C07310=1132.856,310.921,-76.435,-177.796,10.546,149.531
C07311=1132.851,311.169,-76.468,-177.793,10.548,149.531
C07312=1132.848,311.417,-76.500,-177.790,10.550,149.530
C07313=1132.844,311.665,-76.533,-177.787,10.553,149.530
C07314=1132.839,311.913,-76.564,-177.783,10.556,149.530
C07315=1132.835,312.160,-76.597,-177.780,10.558,149.530
C07316=1132.831,312.408,-76.629,-177.777,10.561,149.530
C07317=1132.827,312.656,-76.662,-177.774,10.563,149.529
C07318=1132.824,312.904,-76.694,-177.771,10.566,149.529
C07319=1132.820,313.152,-76.727,-177.767,10.569,149.529
C07320=1132.815,313.400,-76.760,-177.765,10.571,149.529
C07321=1132.812,313.648,-76.792,-177.761,10.574,149.529
C07322=1132.807,313.895,-76.824,-177.758,10.576,149.529
C07323=1132.803,314.143,-76.857,-177.755,10.579,149.529
C07324=1132.799,314.391,-76.889,-177.752,10.581,149.528
C07325=1132.795,314.639,-76.923,-177.749,10.584,149.528
C07326=1132.791,314.887,-76.954,-177.745,10.587,149.528
C07327=1132.787,315.134,-76.988,-177.742,10.589,149.528
C07328=1132.782,315.383,-77.020,-177.739,10.592,149.528
C07329=1132.779,315.630,-77.053,-177.736,10.594,149.527
C07330=1132.775,315.878,-77.086,-177.733,10.596,149.527
C07331=1132.770,316.126,-77.118,-177.730,10.599,149.527
C07332=1132.767,316.374,-77.151,-177.727,10.601,149.527
C07333=1132.763,316.621,-77.184,-177.724,10.604,149.527
C07334=1132.758,316.870,-77.216,-177.721,10.606,149.526
C07335=1132.754,317.118,-77.249,-177.717,10.609,149.526
C07336=1132.751,317.365,-77.282,-177.714,10.612,149.526
C07337=1132.746,317.613,-77.314,-177.711,10.614,149.526
C07338=1132.742,317.861,-77.348,-177.708,10.616,149.526
C07339=1132.738,318.109,-77.381,-177.705,10.619,149.525
C07340=1132.735,318.356,-77.413,-177.701,10.622,149.525
C07341=1132.730,318.605,-77.446,-177.698,10.624,149.525
C07342=1132.726,318.852,-77.479,-177.695,10.627,149.525
C07343=1132.722,319.100,-77.512,-177.692,10.629,149.525
C07344=1132.719,319.347,-77.545,-177.689,10.632,149.525
C07345=1132.714,319.595,-77.578,-177.686,10.635,149.524
C07346=1132.710,319.843,-77.611,-177.682,10.637,149.524
C07347=1132.706,320.091,-77.643,-177.679,10.640,149.524
C07348=1132.702,320.339,-77.677,-177.676,10.642,149.524
C07349=1132.698,320.587,-77.710,-177.673,10.645,149.524
C07350=1132.695,320.799,-77.738,-177.670,10.647,149.523
C07351=1132.691,321.013,-77.766,-177.668,10.648,149.523
C07352=1132.687,321.226,-77.794,-177.665,10.651,149.523
C07353=1132.684,321.440,-77.824,-177.662,10.653,149.523
C07354=1132.680,321.653,-77.852,-177.659,10.655,149.523
C07355=1132.677,321.866,-77.881,-177.657,10.657,149.523
C07356=1132.673,322.080,-77.909,-177.654,10.659,149.522
C07357=1132.671,322.293,-77.937,-177.651,10.662,149.522
C07358=1132.667,322.541,-77.971,-177.648,10.664,149.522
C07359=1132.663,322.788,-78.004,-177.645,10.667,149.522
C07360=1132.658,323.036,-78.037,-177.642,10.670,149.522
C07361=1132.654,323.284,-78.070,-177.638,10.672,149.521
C07362=1132.650,323.532,-78.103,-177.635,10.675,149.521
C07363=1132.646,323.779,-78.136,-177.632,10.677,149.521
C07364=1132.642,324.027,-78.170,-177.629,10.680,149.521
C07365=1132.638,324.276,-78.203,-177.625,10.682,149.521
C07366=1132.634,324.523,-78.236,-177.623,10.684,149.521
C07367=1132.630,324.770,-78.270,-177.620,10.687,149.520
C07368=1132.626,325.018,-78.303,-177.616,10.689,149.520
C07369=1132.622,325.266,-78.336,-177.614,10.692,149.520
C07370=1132.618,325.514,-78.370,-177.610,10.694,149.520
C07371=1132.614,325.761,-78.403,-177.607,10.697,149.520
C07372=1132.610,326.010,-78.436,-177.604,10.699,149.519
C07373=1132.606,326.257,-78.470,-177.601,10.702,149.519
C07374=1132.602,326.505,-78.503,-177.597,10.704,149.519
C07375=1132.598,326.752,-78.536,-177.594,10.707,149.519
C07376=1132.594,327.000,-78.570,-177.591,10.710,149.519
C07377=1132.590,327.247,-78.603,-177.588,10.712,149.518
C07378=1132.586,327.496,-78.638,-177.584,10.714,149.518
C07379=1132.582,327.744,-78.671,-177.582,10.717,149.518
C07380=1132.578,327.991,-78.705,-177.578,10.720,149.518
C07381=1132.574,328.238,-78.738,-177.575,10.722,149.518
C07382=1132.570,328.486,-78.771,-177.572,10.725,149.518
C07383=1132.566,328.734,-78.805,-177.569,10.727,149.517
C07384=1132.562,328.982,-78.838,-177.565,10.730,149.517
C07385=1132.557,329.230,-78.872,-177.562,10.732,149.517
C07386=1132.554,329.477,-78.906,-177.559,10.735,149.517
C07387=1132.550,329.725,-78.939,-177.556,10.737,149.516
C07388=1132.546,329.972,-78.973,-177.552,10.740,149.516
C07389=1132.542,330.220,-79.007,-177.549,10.743,149.516
C07390=1132.538,330.467,-79.040,-177.546,10.745,149.516
C07391=1132.534,330.716,-79.074,-177.543,10.748,149.516
C07392=1132.530,330.963,-79.108,-177.540,10.749,149.515
C07393=1132.526,331.211,-79.142,-177.537,10.752,149.515
C07394=1132.522,331.458,-79.175,-177.534,10.754,149.515
C07395=1132.518,331.707,-79.210,-177.531,10.757,149.515
C07396=1132.514,331.954,-79.243,-177.527,10.759,149.515
C07397=1132.510,332.202,-79.277,-177.524,10.762,149.515
C07398=1132.507,332.449,-79.311,-177.521,10.765,149.514
C07399=1132.502,332.697,-79.345,-177.518,10.767,149.514
C07400=1132.498,332.944,-79.378,-177.514,10.769,149.514
C07401=1132.495,333.192,-79.413,-177.511,10.772,149.514
C07402=1132.490,333.440,-79.446,-177.508,10.775,149.514
C07403=1132.486,333.687,-79.480,-177.505,10.777,149.513
C07404=1132.483,333.935,-79.514,-177.501,10.780,149.513
C07405=1132.478,334.183,-79.548,-177.499,10.782,149.513
C07406=1132.474,334.396,-79.577,-177.496,10.784,149.513
C07407=1132.472,334.609,-79.607,-177.493,10.787,149.513
C07408=1132.468,334.822,-79.636,-177.490,10.789,149.512
C07409=1132.465,335.036,-79.666,-177.487,10.791,149.512
C07410=1132.461,335.249,-79.695,-177.485,10.793,149.512
C07411=1132.458,335.462,-79.724,-177.481,10.795,149.512
C07412=1132.454,335.676,-79.753,-177.479,10.797,149.512
C07413=1132.450,335.888,-79.782,-177.476,10.799,149.511
C07414=1132.447,336.136,-79.817,-177.473,10.802,149.511
C07415=1132.443,336.384,-79.851,-177.470,10.804,149.511
C07416=1132.439,336.632,-79.885,-177.467,10.807,149.511
C07417=1132.435,336.879,-79.920,-177.463,10.809,149.511
C07418=1132.431,337.126,-79.954,-177.460,10.812,149.510
C07419=1132.427,337.374,-79.987,-177.457,10.814,149.510
C07420=1132.423,337.622,-80.022,-177.454,10.817,149.510
C07421=1132.420,337.870,-80.056,-177.451,10.819,149.510
C07422=1132.415,338.117,-80.090,-177.447,10.822,149.510
C07423=1132.412,338.365,-80.125,-177.444,10.825,149.510
C07424=1132.407,338.612,-80.159,-177.441,10.827,149.509
C07425=1132.403,338.859,-80.193,-177.438,10.830,149.509
C07426=1132.400,339.108,-80.228,-177.434,10.832,149.509
C07427=1132.396,339.355,-80.262,-177.431,10.834,149.509
C07428=1132.392,339.603,-80.296,-177.428,10.837,149.508
C07429=1132.387,339.850,-80.331,-177.425,10.840,149.508
C07430=1132.384,340.098,-80.365,-177.422,10.842,149.508
C07431=1132.379,340.345,-80.400,-177.418,10.845,149.508
C07432=1132.376,340.593,-80.434,-177.415,10.847,149.508
C07433=1132.372,340.841,-80.468,-177.412,10.849,149.507
C07434=1132.368,341.088,-80.502,-177.409,10.852,149.507
C07435=1132.364,341.336,-80.537,-177.405,10.855,149.507
C07436=1132.359,341.583,-80.571,-177.402,10.857,149.507
C07437=1132.356,341.831,-80.606,-177.399,10.860,149.507
C07438=1132.352,342.078,-80.641,-177.395,10.862,149.506
C07439=1132.348,342.326,-80.676,-177.392,10.865,149.506
C07440=1132.344,342.573,-80.710,-177.389,10.867,149.506
C07441=1132.340,342.821,-80.744,-177.386,10.870,149.506
C07442=1132.335,343.069,-80.779,-177.383,10.872,149.506
C07443=1132.332,343.316,-80.814,-177.379,10.875,149.506
C07444=1132.328,343.564,-80.849,-177.377,10.876,149.505
C07445=1132.324,343.811,-80.883,-177.373,10.879,149.505
C07446=1132.321,344.059,-80.917,-177.370,10.882,149.505
C07447=1132.316,344.306,-80.953,-177.367,10.884,149.505
C07448=1132.312,344.554,-80.987,-177.364,10.887,149.505
C07449=1132.308,344.802,-81.022,-177.360,10.889,149.504
C07450=1132.305,345.049,-81.057,-177.357,10.891,149.504
C07451=1132.300,345.296,-81.091,-177.354,10.894,149.504
C07452=1132.296,345.544,-81.126,-177.350,10.896,149.504
C07453=1132.293,345.792,-81.162,-177.348,10.899,149.504
C07454=1132.289,346.039,-81.196,-177.344,10.902,149.503
C07455=1132.285,346.287,-81.230,-177.341,10.904,149.503
C07456=1132.281,346.534,-81.266,-177.338,10.907,149.503
C07457=1132.277,346.782,-81.300,-177.334,10.909,149.503
C07458=1132.273,347.030,-81.336,-177.331,10.911,149.502
C07459=1132.269,347.277,-81.370,-177.328,10.914,149.502
C07460=1132.266,347.524,-81.405,-177.324,10.916,149.502
C07461=1132.262,347.772,-81.440,-177.321,10.919,149.502
C07462=1132.258,347.985,-81.470,-177.319,10.921,149.502
C07463=1132.255,348.198,-81.500,-177.315,10.923,149.501
C07464=1132.251,348.412,-81.530,-177.313,10.925,149.501
C07465=1132.247,348.624,-81.560,-177.310,10.928,149.501
C07466=1132.244,348.838,-81.591,-177.307,10.929,149.501
C07467=1132.241,349.050,-81.621,-177.304,10.932,149.501
C07468=1132.237,349.263,-81.651,-177.302,10.934,149.501
C07469=1132.234,349.476,-81.682,-177.299,10.936,149.500
C07470=1132.230,349.724,-81.716,-177.295,10.939,149.500
C07471=1132.227,349.971,-81.751,-177.292,10.941,149.500
C07472=1132.223,350.218,-81.787,-177.288,10.945,149.500
C07473=1132.219,350.467,-81.821,-177.284,10.947,149.499
C07474=1132.215,350.713,-81.857,-177.280,10.950,149.499
C07475=1132.211,350.961,-81.892,-177.277,10.952,149.499
C07476=1132.207,351.209,-81.927,-177.273,10.956,149.499
C07477=1132.203,351.456,-81.963,-177.269,10.958,149.498
C07478=1132.199,351.703,-81.998,-177.266,10.960,149.498
C07479=1132.195,351.951,-82.033,-177.262,10.963,149.498
C07480=1132.192,352.199,-82.068,-177.258,10.966,149.497
C07481=1132.187,352.446,-82.103,-177.255,10.968,149.497
C07482=1132.184,352.693,-82.139,-177.251,10.971,149.497
C07483=1132.180,352.941,-82.174,-177.248,10.974,149.497
C07484=1132.176,353.189,-82.209,-177.243,10.977,149.496
C07485=1132.172,353.436,-82.245,-177.240,10.979,149.496
C07486=1132.168,353.683,-82.280,-177.237,10.982,149.496
C07487=1132.164,353.931,-82.315,-177.233,10.984,149.495
C07488=1132.161,354.178,-82.351,-177.229,10.987,149.495
C07489=1132.157,354.426,-82.387,-177.226,10.989,149.495
C07490=1132.152,354.673,-82.422,-177.222,10.992,149.495
C07491=1132.148,354.920,-82.458,-177.218,10.995,149.494
C07492=1132.145,355.168,-82.493,-177.215,10.997,149.494
C07493=1132.141,355.415,-82.529,-177.211,11.000,149.494
C07494=1132.137,355.663,-82.565,-177.208,11.002,149.494
C07495=1132.134,355.910,-82.600,-177.204,11.004,149.493
C07496=1132.129,356.157,-82.635,-177.200,11.008,149.493
C07497=1132.126,356.405,-82.671,-177.197,11.010,149.493
C07498=1132.121,356.652,-82.707,-177.193,11.012,149.493
C07499=1132.118,356.900,-82.743,-177.190,11.015,149.492
C07500=1132.114,357.147,-82.778,-177.187,11.017,149.492
C07501=1132.110,357.395,-82.814,-177.182,11.020,149.492
C07502=1132.107,357.642,-82.849,-177.179,11.022,149.492
C07503=1132.102,357.890,-82.885,-177.176,11.025,149.491
C07504=1132.098,358.137,-82.920,-177.172,11.027,149.491
C07505=1132.094,358.384,-82.956,-177.169,11.030,149.491
C07506=1132.091,358.631,-82.992,-177.166,11.032,149.491
C07507=1132.087,358.879,-83.028,-177.162,11.034,149.490
C07508=1132.083,359.127,-83.064,-177.158,11.037,149.490
C07509=1132.079,359.374,-83.100,-177.155,11.039,149.490
C07510=1132.076,359.622,-83.135,-177.151,11.042,149.489
C07511=1132.072,359.869,-83.172,-177.148,11.044,149.489
C07512=1132.068,360.116,-83.207,-177.144,11.047,149.489
C07513=1132.064,360.364,-83.243,-177.141,11.049,149.489
C07514=1132.061,360.611,-83.279,-177.138,11.052,149.488
C07515=1132.057,360.859,-83.315,-177.134,11.054,149.488
C07516=1132.053,361.106,-83.351,-177.131,11.056,149.488
C07517=1132.049,361.353,-83.387,-177.127,11.059,149.488
C07518=1132.045,361.566,-83.418,-177.125,11.061,149.487
C07519=1132.042,361.778,-83.449,-177.121,11.063,149.487
C07520=1132.038,361.992,-83.480,-177.119,11.065,149.487
C07521=1132.035,362.204,-83.511,-177.115,11.067,149.487
C07522=1132.032,362.418,-83.542,-177.113,11.069,149.486
C07523=1132.029,362.630,-83.573,-177.110,11.071,149.486
C07524=1132.026,362.843,-83.604,-177.107,11.073,149.486
C07525=1132.023,363.056,-83.635,-177.104,11.075,149.486
C07526=1132.018,363.303,-83.672,-177.101,11.078,149.486
C07527=1132.015,363.551,-83.707,-177.097,11.080,149.485
C07528=1132.011,363.798,-83.744,-177.094,11.082,149.485
C07529=1132.007,364.046,-83.780,-177.091,11.085,149.485
C07530=1132.004,364.293,-83.816,-177.088,11.087,149.485
C07531=1131.999,364.540,-83.852,-177.084,11.090,149.484
C07532=1131.996,364.787,-83.888,-177.081,11.092,149.484
C07533=1131.992,365.035,-83.924,-177.078,11.093,149.484
C07534=1131.988,365.282,-83.961,-177.075,11.096,149.484
C07535=1131.984,365.529,-83.998,-177.071,11.098,149.483
C07536=1131.980,365.777,-84.033,-177.068,11.101,149.483
C07537=1131.976,366.024,-84.070,-177.065,11.103,149.483
C07538=1131.973,366.272,-84.106,-177.061,11.106,149.483
C07539=1131.969,366.519,-84.143,-177.058,11.108,149.482
C07540=1131.966,366.766,-84.179,-177.055,11.110,149.482
C07541=1131.961,367.014,-84.215,-177.052,11.112,149.482
C07542=1131.958,367.261,-84.251,-177.049,11.115,149.482
C07543=1131.954,367.508,-84.288,-177.045,11.117,149.482
C07544=1131.951,367.755,-84.325,-177.042,11.120,149.481
C07545=1131.946,368.003,-84.361,-177.039,11.121,149.481
C07546=1131.942,368.250,-84.398,-177.036,11.124,149.481
C07547=1131.939,368.497,-84.434,-177.032,11.126,149.481
C07548=1131.935,368.744,-84.471,-177.029,11.129,149.480
C07549=1131.932,368.992,-84.507,-177.026,11.131,149.480
C07550=1131.927,369.239,-84.543,-177.023,11.133,149.480
C07551=1131.923,369.486,-84.580,-177.020,11.136,149.480
C07552=1131.920,369.733,-84.617,-177.017,11.138,149.480
C07553=1131.916,369.981,-84.653,-177.014,11.141,149.479
C07554=1131.912,370.228,-84.690,-177.011,11.142,149.479
C07555=1131.908,370.475,-84.726,-177.008,11.145,149.479
C07556=1131.905,370.723,-84.763,-177.004,11.147,149.479
C07557=1131.901,370.970,-84.800,-177.002,11.149,149.478
C07558=1131.897,371.217,-84.836,-176.998,11.151,149.478
C07559=1131.893,371.464,-84.873,-176.995,11.154,149.478
C07560=1131.889,371.712,-84.910,-176.992,11.156,149.478
C07561=1131.886,371.958,-84.946,-176.989,11.158,149.478
C07562=1131.882,372.206,-84.983,-176.986,11.161,149.478
C07563=1131.878,372.454,-85.020,-176.984,11.163,149.477
C07564=1131.874,372.701,-85.057,-176.980,11.165,149.477
C07565=1131.871,372.948,-85.093,-176.977,11.167,149.477
C07566=1131.867,373.195,-85.130,-176.974,11.169,149.477
C07567=1131.863,373.443,-85.167,-176.971,11.172,149.477
C07568=1131.859,373.690,-85.204,-176.968,11.174,149.476
C07569=1131.856,373.937,-85.241,-176.965,11.176,149.476
C07570=1131.852,374.184,-85.277,-176.962,11.179,149.476
C07571=1131.848,374.432,-85.315,-176.959,11.181,149.476
C07572=1131.844,374.679,-85.352,-176.957,11.183,149.476
C07573=1131.840,374.926,-85.388,-176.953,11.186,149.476
C07574=1131.837,375.138,-85.420,-176.951,11.188,149.475
C07575=1131.833,375.351,-85.452,-176.948,11.189,149.475
C07576=1131.830,375.564,-85.484,-176.946,11.191,149.475
C07577=1131.827,375.778,-85.516,-176.944,11.193,149.475
C07578=1131.824,375.990,-85.548,-176.941,11.195,149.475
C07579=1131.821,376.203,-85.580,-176.939,11.197,149.475
C07580=1131.818,376.415,-85.611,-176.937,11.199,149.475
C07581=1131.814,376.628,-85.643,-176.934,11.201,149.475
C07582=1131.811,376.874,-85.680,-176.931,11.204,149.474
C07583=1131.807,377.122,-85.717,-176.928,11.206,149.474
C07584=1131.803,377.370,-85.754,-176.925,11.208,149.474
C07585=1131.799,377.616,-85.791,-176.922,11.211,149.474
C07586=1131.796,377.864,-85.829,-176.920,11.213,149.474
C07587=1131.792,378.111,-85.865,-176.917,11.215,149.474
C07588=1131.788,378.358,-85.902,-176.914,11.217,149.474
C07589=1131.784,378.605,-85.940,-176.911,11.220,149.474
C07590=1131.780,378.853,-85.977,-176.909,11.222,149.473
C07591=1131.776,379.100,-86.014,-176.905,11.224,149.473
C07592=1131.772,379.347,-86.052,-176.903,11.226,149.473
C07593=1131.769,379.594,-86.089,-176.900,11.229,149.473
C07594=1131.765,379.842,-86.126,-176.898,11.231,149.473
C07595=1131.761,380.088,-86.163,-176.895,11.234,149.473
C07596=1131.758,380.336,-86.200,-176.892,11.236,149.473
C07597=1131.755,380.582,-86.237,-176.889,11.238,149.473
C07598=1131.750,380.830,-86.274,-176.887,11.240,149.473
C07599=1131.747,381.077,-86.311,-176.884,11.243,149.473
C07600=1131.742,381.324,-86.350,-176.882,11.245,149.473
C07601=1131.739,381.572,-86.387,-176.878,11.247,149.472
C07602=1131.735,381.819,-86.424,-176.876,11.249,149.472
C07603=1131.731,382.066,-86.461,-176.873,11.252,149.472
C07604=1131.728,382.313,-86.499,-176.871,11.254,149.472
C07605=1131.724,382.560,-86.536,-176.868,11.257,149.472
C07606=1131.720,382.807,-86.574,-176.866,11.259,149.472
C07607=1131.716,383.055,-86.611,-176.863,11.261,149.472
C07608=1131.713,383.301,-86.648,-176.861,11.264,149.472
C07609=1131.710,383.549,-86.686,-176.858,11.266,149.472
C07610=1131.705,383.796,-86.723,-176.857,11.268,149.472
C07611=1131.702,384.043,-86.761,-176.856,11.269,149.472
C07612=1131.698,384.290,-86.798,-176.855,11.271,149.472
C07613=1131.694,384.537,-86.836,-176.853,11.272,149.472
C07614=1131.691,384.785,-86.873,-176.852,11.274,149.473
C07615=1131.687,385.031,-86.910,-176.851,11.276,149.473
C07616=1131.683,385.279,-86.949,-176.850,11.277,149.473
C07617=1131.679,385.526,-86.986,-176.849,11.279,149.473
C07618=1131.675,385.773,-87.023,-176.848,11.281,149.473
C07619=1131.672,386.021,-87.061,-176.847,11.282,149.473
C07620=1131.668,386.267,-87.098,-176.846,11.284,149.474
C07621=1131.665,386.515,-87.136,-176.845,11.286,149.474
C07622=1131.661,386.762,-87.173,-176.844,11.288,149.474
C07623=1131.658,387.009,-87.211,-176.842,11.289,149.474
C07624=1131.654,387.256,-87.249,-176.842,11.291,149.474
C07625=1131.649,387.504,-87.286,-176.841,11.293,149.475
C07626=1131.646,387.750,-87.324,-176.839,11.295,149.475
C07627=1131.642,387.997,-87.362,-176.839,11.297,149.475
C07628=1131.638,388.245,-87.399,-176.838,11.298,149.475
C07629=1131.635,388.491,-87.436,-176.837,11.300,149.475
C07630=1131.632,388.704,-87.469,-176.836,11.302,149.476
C07631=1131.628,388.917,-87.502,-176.835,11.304,149.476
C07632=1131.625,389.129,-87.533,-176.834,11.306,149.476
C07633=1131.622,389.342,-87.566,-176.834,11.307,149.476
C07634=1131.619,389.555,-87.599,-176.833,11.309,149.477
C07635=1131.615,389.767,-87.631,-176.832,11.311,149.477
C07636=1131.613,389.979,-87.663,-176.831,11.313,149.477
C07637=1131.609,390.193,-87.695,-176.831,11.314,149.477
C07638=1131.606,390.439,-87.733,-176.829,11.316,149.478
C07639=1131.602,390.687,-87.772,-176.829,11.318,149.478
C07640=1131.598,390.934,-87.809,-176.828,11.320,149.478
C07641=1131.594,391.181,-87.846,-176.827,11.322,149.479
C07642=1131.591,391.428,-87.884,-176.827,11.325,149.479
C07643=1131.588,391.675,-87.922,-176.826,11.327,149.479
C07644=1131.584,391.922,-87.959,-176.825,11.329,149.480
C07645=1131.579,392.170,-87.997,-176.825,11.331,149.480
C07646=1131.576,392.417,-88.035,-176.824,11.333,149.481
C07647=1131.573,392.664,-88.073,-176.824,11.335,149.481
C07648=1131.569,392.910,-88.110,-176.823,11.337,149.481
C07649=1131.566,393.158,-88.148,-176.822,11.340,149.482
C07650=1131.561,393.405,-88.186,-176.821,11.342,149.482
C07651=1131.557,393.652,-88.223,-176.821,11.344,149.483
C07652=1131.554,393.899,-88.261,-176.820,11.347,149.483
C07653=1131.550,394.146,-88.299,-176.820,11.349,149.484
C07654=1131.546,394.393,-88.337,-176.819,11.351,149.484
C07655=1131.542,394.640,-88.375,-176.819,11.353,149.485
C07656=1131.539,394.888,-88.412,-176.818,11.356,149.485
C07657=1131.536,395.135,-88.450,-176.817,11.359,149.486
C07658=1131.531,395.382,-88.488,-176.817,11.361,149.486
C07659=1131.528,395.629,-88.526,-176.817,11.363,149.487
C07660=1131.524,395.876,-88.564,-176.816,11.366,149.487
C07661=1131.520,396.123,-88.602,-176.816,11.368,149.488
C07662=1131.516,396.370,-88.640,-176.816,11.370,149.488
C07663=1131.513,396.617,-88.678,-176.815,11.374,149.489
C07664=1131.509,396.864,-88.715,-176.815,11.376,149.489
C07665=1131.505,397.112,-88.753,-176.815,11.379,149.490
C07666=1131.501,397.358,-88.791,-176.815,11.381,149.491
C07667=1131.498,397.606,-88.829,-176.814,11.383,149.491
C07668=1131.494,397.852,-88.866,-176.814,11.386,149.492
C07669=1131.490,398.100,-88.905,-176.813,11.389,149.493
C07670=1131.487,398.346,-88.942,-176.813,11.392,149.493
C07671=1131.483,398.594,-88.980,-176.813,11.394,149.494
C07672=1131.479,398.841,-89.019,-176.813,11.397,149.495
C07673=1131.476,399.088,-89.056,-176.813,11.399,149.495
C07674=1131.472,399.334,-89.094,-176.812,11.403,149.496
C07675=1131.468,399.582,-89.133,-176.813,11.406,149.497
C07676=1131.465,399.829,-89.171,-176.813,11.408,149.497
C07677=1131.461,400.076,-89.208,-176.813,11.411,149.498
C07678=1131.457,400.323,-89.247,-176.812,11.414,149.499
C07679=1131.453,400.570,-89.284,-176.812,11.417,149.499
C07680=1131.450,400.817,-89.322,-176.812,11.420,149.500
C07681=1131.445,401.065,-89.360,-176.812,11.422,149.501
C07682=1131.442,401.312,-89.398,-176.812,11.426,149.502
C07683=1131.438,401.559,-89.435,-176.812,11.429,149.502
C07684=1131.434,401.806,-89.474,-176.812,11.432,149.503
C07685=1131.432,402.053,-89.512,-176.812,11.435,149.504
C07686=1131.428,402.265,-89.545,-176.812,11.438,149.505
C07687=1131.425,402.478,-89.577,-176.812,11.441,149.506
C07688=1131.422,402.691,-89.610,-176.812,11.443,149.506
C07689=1131.419,402.903,-89.642,-176.813,11.446,149.507
C07690=1131.415,403.115,-89.675,-176.812,11.449,149.508
C07691=1131.413,403.328,-89.708,-176.813,11.452,149.509
C07692=1131.409,403.540,-89.741,-176.813,11.454,149.509
C07693=1131.406,403.753,-89.773,-176.813,11.457,149.510
C07694=1131.402,404.000,-89.811,-176.813,11.460,149.511
C07695=1131.399,404.248,-89.850,-176.814,11.463,149.512
C07696=1131.395,404.494,-89.887,-176.814,11.467,149.513
C07697=1131.391,404.742,-89.926,-176.814,11.470,149.514
C07698=1131.387,404.988,-89.963,-176.815,11.473,149.515
C07699=1131.384,405.236,-90.001,-176.815,11.477,149.516
C07700=1131.380,405.482,-90.040,-176.816,11.480,149.517
C07701=1131.376,405.729,-90.078,-176.816,11.483,149.518
C07702=1131.373,405.976,-90.116,-176.816,11.487,149.519
C07703=1131.369,406.223,-90.154,-176.817,11.490,149.520
C07704=1131.366,406.471,-90.192,-176.817,11.494,149.521
C07705=1131.361,406.717,-90.230,-176.817,11.497,149.522
C07706=1131.358,406.965,-90.268,-176.818,11.502,149.523
C07707=1131.355,407.212,-90.306,-176.819,11.505,149.524
C07708=1131.350,407.459,-90.344,-176.819,11.508,149.525
C07709=1131.347,407.706,-90.382,-176.819,11.512,149.526
C07710=1131.343,407.953,-90.422,-176.820,11.516,149.527
C07711=1131.340,408.200,-90.459,-176.821,11.520,149.528
C07712=1131.336,408.447,-90.497,-176.822,11.523,149.529
C07713=1131.332,408.694,-90.535,-176.822,11.527,149.531
C07714=1131.329,408.941,-90.573,-176.823,11.531,149.532
C07715=1131.325,409.189,-90.612,-176.823,11.535,149.533
C07716=1131.321,409.435,-90.649,-176.824,11.539,149.534
C07717=1131.317,409.682,-90.689,-176.824,11.543,149.535
C07718=1131.314,409.929,-90.726,-176.825,11.546,149.536
C07719=1131.310,410.176,-90.764,-176.826,11.551,149.538
C07720=1131.306,410.424,-90.803,-176.826,11.555,149.539
C07721=1131.303,410.670,-90.840,-176.828,11.559,149.540
C07722=1131.299,410.917,-90.879,-176.828,11.563,149.542
C07723=1131.296,411.164,-90.917,-176.829,11.567,149.543
C07724=1131.291,411.411,-90.955,-176.830,11.571,149.544
C07725=1131.288,411.659,-90.993,-176.831,11.575,149.545
C07726=1131.284,411.906,-91.032,-176.832,11.579,149.547
C07727=1131.281,412.152,-91.070,-176.833,11.584,149.548
C07728=1131.277,412.400,-91.109,-176.834,11.588,149.549
C07729=1131.274,412.647,-91.147,-176.835,11.592,149.551
C07730=1131.270,412.893,-91.184,-176.836,11.596,149.552
C07731=1131.266,413.141,-91.223,-176.837,11.600,149.553
C07732=1131.262,413.387,-91.261,-176.838,11.605,149.555
C07733=1131.258,413.635,-91.300,-176.839,11.609,149.556
C07734=1131.255,413.882,-91.338,-176.840,11.614,149.558
C07735=1131.251,414.129,-91.376,-176.841,11.619,149.559
C07736=1131.248,414.375,-91.414,-176.842,11.623,149.561
C07737=1131.246,414.623,-91.452,-176.844,11.627,149.562
C07738=1131.243,414.870,-91.491,-176.845,11.632,149.564
C07739=1131.242,415.117,-91.528,-176.846,11.637,149.565
C07740=1131.242,415.364,-91.566,-176.847,11.641,149.567
C07741=1131.241,415.611,-91.604,-176.849,11.646,149.568
C07742=1131.242,415.824,-91.637,-176.850,11.650,149.569
C07743=1131.242,416.036,-91.669,-176.851,11.654,149.571
C07744=1131.244,416.248,-91.702,-176.852,11.658,149.572
C07745=1131.246,416.461,-91.734,-176.854,11.662,149.574
C07746=1131.247,416.673,-91.766,-176.855,11.666,149.575
C07747=1131.250,416.885,-91.798,-176.856,11.670,149.576
C07748=1131.253,417.098,-91.830,-176.857,11.674,149.578
C07749=1131.257,417.310,-91.861,-176.859,11.678,149.579
C07750=1130.838,417.310,-91.924,-176.851,11.683,149.578
C07751=1130.834,417.097,-91.893,-176.850,11.679,149.577
C07752=1130.831,416.885,-91.860,-176.848,11.675,149.576
C07753=1130.828,416.673,-91.828,-176.847,11.671,149.574
C07754=1130.826,416.460,-91.796,-176.846,11.666,149.573
C07755=1130.824,416.248,-91.764,-176.845,11.662,149.571
C07756=1130.823,416.036,-91.732,-176.844,11.658,149.570
C07757=1130.822,415.823,-91.699,-176.843,11.654,149.569
C07758=1130.822,415.611,-91.667,-176.841,11.650,149.567
C07759=1130.822,415.364,-91.628,-176.840,11.645,149.566
C07760=1130.823,415.117,-91.591,-176.839,11.641,149.564
C07761=1130.824,414.870,-91.554,-176.838,11.636,149.563
C07762=1130.826,414.623,-91.515,-176.837,11.632,149.561
C07763=1130.829,414.376,-91.476,-176.836,11.627,149.560
C07764=1130.832,414.129,-91.439,-176.835,11.622,149.558
C07765=1130.836,413.881,-91.400,-176.834,11.617,149.557
C07766=1130.840,413.635,-91.362,-176.832,11.614,149.556
C07767=1130.843,413.388,-91.323,-176.831,11.609,149.554
C07768=1130.846,413.140,-91.285,-176.831,11.604,149.553
C07769=1130.851,412.893,-91.247,-176.829,11.600,149.551
C07770=1130.854,412.647,-91.208,-176.829,11.596,149.550
C07771=1130.857,412.400,-91.170,-176.828,11.591,149.549
C07772=1130.861,412.153,-91.132,-176.827,11.587,149.547
C07773=1130.865,411.905,-91.094,-176.826,11.583,149.546
C07774=1130.869,411.658,-91.056,-176.825,11.579,149.545
C07775=1130.872,411.412,-91.018,-176.825,11.574,149.543
C07776=1130.876,411.164,-90.979,-176.823,11.570,149.542
C07777=1130.879,410.917,-90.941,-176.823,11.566,149.541
C07778=1130.884,410.670,-90.903,-176.822,11.563,149.540
C07779=1130.887,410.423,-90.864,-176.821,11.558,149.538
C07780=1130.890,410.176,-90.826,-176.821,11.554,149.537
C07781=1130.894,409.929,-90.788,-176.820,11.550,149.536
C07782=1130.898,409.682,-90.750,-176.819,11.546,149.535
C07783=1130.902,409.435,-90.712,-176.818,11.542,149.534
C07784=1130.905,409.189,-90.673,-176.818,11.538,149.532
C07785=1130.909,408.941,-90.635,-176.817,11.534,149.531
C07786=1130.913,408.694,-90.597,-176.816,11.531,149.530
C07787=1130.916,408.447,-90.559,-176.816,11.526,149.529
C07788=1130.920,408.200,-90.521,-176.815,11.523,149.528
C07789=1130.924,407.953,-90.483,-176.815,11.519,149.527
C07790=1130.927,407.706,-90.444,-176.814,11.516,149.526
C07791=1130.931,407.459,-90.406,-176.814,11.512,149.524
C07792=1130.935,407.212,-90.368,-176.813,11.508,149.523
C07793=1130.938,406.965,-90.330,-176.813,11.504,149.522
C07794=1130.943,406.718,-90.292,-176.812,11.501,149.521
C07795=1130.946,406.470,-90.254,-176.812,11.497,149.520
C07796=1130.949,406.223,-90.216,-176.811,11.494,149.519
C07797=1130.953,405.976,-90.178,-176.812,11.490,149.518
C07798=1130.956,405.730,-90.139,-176.811,11.487,149.517
C07799=1130.961,405.483,-90.101,-176.811,11.483,149.516
C07800=1130.964,405.235,-90.063,-176.810,11.480,149.515
C07801=1130.967,404.988,-90.025,-176.810,11.476,149.514
C07802=1130.972,404.741,-89.987,-176.810,11.473,149.513
C07803=1130.975,404.494,-89.949,-176.809,11.470,149.512
C07804=1130.979,404.247,-89.911,-176.809,11.466,149.511
C07805=1130.983,404.000,-89.873,-176.809,11.463,149.511
C07806=1130.986,403.753,-89.835,-176.809,11.459,149.510
C07807=1130.989,403.540,-89.802,-176.809,11.456,149.509
C07808=1130.993,403.328,-89.770,-176.809,11.453,149.508
C07809=1130.995,403.115,-89.736,-176.809,11.451,149.507
C07810=1130.999,402.903,-89.703,-176.808,11.448,149.507
C07811=1131.002,402.691,-89.671,-176.809,11.445,149.506
C07812=1131.005,402.478,-89.638,-176.809,11.443,149.505
C07813=1131.009,402.265,-89.605,-176.808,11.440,149.504
C07814=1131.012,402.053,-89.573,-176.808,11.437,149.504
C07815=1131.015,401.806,-89.535,-176.808,11.435,149.503
C07816=1131.019,401.559,-89.497,-176.808,11.431,149.502
C07817=1131.023,401.312,-89.459,-176.808,11.428,149.501
C07818=1131.026,401.064,-89.421,-176.808,11.425,149.501
C07819=1131.030,400.818,-89.383,-176.809,11.422,149.500
C07820=1131.034,400.570,-89.345,-176.808,11.419,149.499
C07821=1131.038,400.324,-89.307,-176.809,11.417,149.498
C07822=1131.041,400.076,-89.269,-176.809,11.413,149.498
C07823=1131.045,399.830,-89.231,-176.809,11.410,149.497
C07824=1131.049,399.582,-89.193,-176.809,11.408,149.496
C07825=1131.052,399.336,-89.155,-176.809,11.405,149.495
C07826=1131.056,399.088,-89.117,-176.809,11.402,149.495
C07827=1131.060,398.841,-89.079,-176.809,11.399,149.494
C07828=1131.063,398.594,-89.041,-176.810,11.397,149.493
C07829=1131.066,398.347,-89.003,-176.810,11.394,149.493
C07830=1131.071,398.100,-88.965,-176.810,11.391,149.492
C07831=1131.074,397.853,-88.927,-176.811,11.388,149.492
C07832=1131.078,397.606,-88.890,-176.811,11.386,149.491
C07833=1131.082,397.359,-88.851,-176.811,11.383,149.490
C07834=1131.086,397.112,-88.814,-176.812,11.380,149.490
C07835=1131.089,396.864,-88.776,-176.812,11.378,149.489
C07836=1131.094,396.617,-88.738,-176.812,11.375,149.489
C07837=1131.097,396.370,-88.700,-176.813,11.373,149.488
C07838=1131.101,396.123,-88.663,-176.813,11.370,149.487
C07839=1131.104,395.876,-88.625,-176.814,11.367,149.487
C07840=1131.108,395.629,-88.587,-176.814,11.365,149.487
C07841=1131.112,395.382,-88.549,-176.814,11.363,149.486
C07842=1131.115,395.136,-88.511,-176.815,11.360,149.485
C07843=1131.119,394.888,-88.473,-176.816,11.357,149.485
C07844=1131.123,394.640,-88.435,-176.816,11.355,149.484
C07845=1131.127,394.393,-88.398,-176.817,11.353,149.484
C07846=1131.130,394.146,-88.360,-176.817,11.351,149.484
C07847=1131.134,393.900,-88.322,-176.818,11.348,149.483
C07848=1131.138,393.652,-88.284,-176.818,11.346,149.483
C07849=1131.141,393.405,-88.246,-176.819,11.343,149.482
C07850=1131.145,393.158,-88.209,-176.820,11.341,149.482
C07851=1131.149,392.911,-88.171,-176.820,11.339,149.481
C07852=1131.152,392.663,-88.133,-176.821,11.337,149.481
C07853=1131.156,392.417,-88.095,-176.821,11.335,149.480
C07854=1131.159,392.170,-88.057,-176.822,11.332,149.480
C07855=1131.164,391.922,-88.020,-176.823,11.330,149.480
C07856=1131.167,391.675,-87.982,-176.824,11.327,149.479
C07857=1131.171,391.428,-87.944,-176.825,11.326,149.479
C07858=1131.175,391.182,-87.907,-176.825,11.323,149.478
C07859=1131.178,390.934,-87.869,-176.826,11.321,149.478
C07860=1131.182,390.687,-87.832,-176.827,11.320,149.478
C07861=1131.186,390.440,-87.794,-176.828,11.318,149.478
C07862=1131.190,390.193,-87.756,-176.828,11.315,149.477
C07863=1131.192,389.980,-87.723,-176.829,11.313,149.477
C07864=1131.196,389.767,-87.692,-176.830,11.312,149.477
C07865=1131.199,389.555,-87.659,-176.831,11.310,149.476
C07866=1131.202,389.342,-87.626,-176.832,11.308,149.476
C07867=1131.205,389.130,-87.594,-176.832,11.307,149.476
C07868=1131.209,388.918,-87.561,-176.833,11.305,149.476
C07869=1131.212,388.705,-87.530,-176.834,11.303,149.475
C07870=1131.215,388.492,-87.497,-176.835,11.301,149.475
C07871=1131.219,388.245,-87.459,-176.836,11.300,149.475
C07872=1131.222,387.998,-87.421,-176.837,11.298,149.475
C07873=1131.226,387.751,-87.384,-176.838,11.296,149.475
C07874=1131.230,387.504,-87.347,-176.839,11.294,149.474
C07875=1131.233,387.257,-87.309,-176.840,11.292,149.474
C07876=1131.237,387.010,-87.272,-176.841,11.291,149.474
C07877=1131.241,386.762,-87.233,-176.842,11.289,149.474
C07878=1131.245,386.515,-87.196,-176.843,11.287,149.474
C07879=1131.249,386.267,-87.159,-176.845,11.285,149.473
C07880=1131.252,386.021,-87.121,-176.846,11.283,149.473
C07881=1131.256,385.774,-87.083,-176.847,11.281,149.473
C07882=1131.260,385.526,-87.046,-176.848,11.279,149.473
C07883=1131.263,385.280,-87.009,-176.849,11.278,149.473
C07884=1131.267,385.032,-86.971,-176.850,11.276,149.473
C07885=1131.271,384.785,-86.934,-176.851,11.275,149.473
C07886=1131.275,384.538,-86.895,-176.852,11.273,149.472
C07887=1131.279,384.291,-86.858,-176.854,11.271,149.472
C07888=1131.282,384.043,-86.820,-176.855,11.270,149.472
C07889=1131.286,383.796,-86.784,-176.856,11.268,149.472
C07890=1131.290,383.550,-86.746,-176.857,11.266,149.472
C07891=1131.293,383.302,-86.709,-176.860,11.264,149.472
C07892=1131.297,383.055,-86.671,-176.862,11.262,149.472
C07893=1131.300,382.808,-86.633,-176.865,11.260,149.472
C07894=1131.304,382.561,-86.596,-176.867,11.258,149.472
C07895=1131.308,382.314,-86.559,-176.870,11.255,149.472
C07896=1131.312,382.066,-86.522,-176.872,11.253,149.472
C07897=1131.315,381.820,-86.484,-176.875,11.250,149.472
C07898=1131.320,381.572,-86.447,-176.878,11.248,149.472
C07899=1131.323,381.325,-86.409,-176.881,11.245,149.472
C07900=1131.327,381.078,-86.372,-176.883,11.243,149.472
C07901=1131.330,380.830,-86.335,-176.886,11.241,149.472
C07902=1131.334,380.584,-86.298,-176.888,11.239,149.473
C07903=1131.338,380.336,-86.261,-176.891,11.236,149.473
C07904=1131.341,380.089,-86.223,-176.894,11.234,149.473
C07905=1131.345,379.842,-86.186,-176.897,11.231,149.473
C07906=1131.350,379.595,-86.149,-176.899,11.229,149.473
C07907=1131.353,379.347,-86.111,-176.902,11.227,149.473
C07908=1131.357,379.100,-86.074,-176.905,11.225,149.473
C07909=1131.361,378.853,-86.037,-176.908,11.222,149.473
C07910=1131.364,378.606,-86.000,-176.910,11.220,149.474
C07911=1131.368,378.359,-85.963,-176.913,11.218,149.474
C07912=1131.372,378.111,-85.926,-176.916,11.216,149.474
C07913=1131.375,377.864,-85.888,-176.919,11.213,149.474
C07914=1131.380,377.617,-85.851,-176.921,11.211,149.474
C07915=1131.384,377.370,-85.814,-176.924,11.209,149.474
C07916=1131.388,377.123,-85.777,-176.927,11.206,149.474
C07917=1131.390,376.876,-85.740,-176.930,11.204,149.474
C07918=1131.394,376.628,-85.703,-176.933,11.202,149.475
C07919=1131.398,376.415,-85.671,-176.936,11.200,149.475
C07920=1131.401,376.203,-85.639,-176.938,11.198,149.475
C07921=1131.405,375.990,-85.607,-176.940,11.196,149.475
C07922=1131.408,375.778,-85.576,-176.943,11.194,149.475
C07923=1131.411,375.564,-85.544,-176.945,11.192,149.475
C07924=1131.414,375.352,-85.512,-176.948,11.190,149.475
C07925=1131.417,375.139,-85.480,-176.950,11.188,149.475
C07926=1131.420,374.926,-85.449,-176.953,11.186,149.476
C07927=1131.425,374.679,-85.412,-176.956,11.184,149.476
C07928=1131.428,374.433,-85.374,-176.959,11.181,149.476
C07929=1131.432,374.185,-85.337,-176.962,11.179,149.476
C07930=1131.435,373.938,-85.301,-176.965,11.177,149.476
C07931=1131.439,373.691,-85.264,-176.968,11.174,149.476
C07932=1131.443,373.444,-85.227,-176.970,11.172,149.477
C07933=1131.447,373.196,-85.190,-176.974,11.170,149.477
C07934=1131.450,372.949,-85.154,-176.977,11.167,149.477
C07935=1131.454,372.702,-85.117,-176.980,11.166,149.477
C07936=1131.458,372.454,-85.080,-176.983,11.163,149.477
C07937=1131.462,372.207,-85.043,-176.986,11.160,149.477
C07938=1131.465,371.960,-85.006,-176.989,11.159,149.478
C07939=1131.469,371.712,-84.970,-176.992,11.156,149.478
C07940=1131.473,371.465,-84.933,-176.995,11.154,149.478
C07941=1131.477,371.218,-84.896,-176.998,11.152,149.478
C07942=1131.481,370.971,-84.860,-177.001,11.149,149.478
C07943=1131.485,370.723,-84.823,-177.004,11.147,149.479
C07944=1131.488,370.476,-84.787,-177.007,11.145,149.479
C07945=1131.492,370.229,-84.750,-177.010,11.143,149.479
C07946=1131.496,369.981,-84.713,-177.013,11.140,149.479
C07947=1131.500,369.735,-84.677,-177.017,11.138,149.479
C07948=1131.504,369.487,-84.640,-177.019,11.136,149.480
C07949=1131.508,369.240,-84.603,-177.023,11.134,149.480
C07950=1131.511,368.993,-84.568,-177.026,11.131,149.480
C07951=1131.515,368.745,-84.530,-177.029,11.129,149.480
C07952=1131.519,368.498,-84.493,-177.032,11.127,149.481
C07953=1131.522,368.251,-84.457,-177.035,11.124,149.481
C07954=1131.527,368.003,-84.421,-177.038,11.122,149.481
C07955=1131.530,367.756,-84.385,-177.042,11.120,149.481
C07956=1131.534,367.509,-84.348,-177.045,11.117,149.481
C07957=1131.538,367.262,-84.312,-177.048,11.115,149.482
C07958=1131.542,367.014,-84.276,-177.051,11.113,149.482
C07959=1131.546,366.767,-84.239,-177.054,11.110,149.482
C07960=1131.549,366.520,-84.202,-177.058,11.108,149.482
C07961=1131.554,366.272,-84.166,-177.061,11.106,149.483
C07962=1131.557,366.025,-84.130,-177.065,11.103,149.483
C07963=1131.561,365.777,-84.093,-177.067,11.102,149.483
C07964=1131.564,365.530,-84.057,-177.071,11.099,149.483
C07965=1131.568,365.283,-84.020,-177.074,11.097,149.484
C07966=1131.572,365.035,-83.985,-177.077,11.094,149.484
C07967=1131.576,364.788,-83.948,-177.080,11.092,149.484
C07968=1131.580,364.541,-83.912,-177.084,11.089,149.484
C07969=1131.584,364.293,-83.876,-177.088,11.087,149.485
C07970=1131.588,364.046,-83.840,-177.091,11.085,149.485
C07971=1131.591,363.799,-83.804,-177.094,11.082,149.485
C07972=1131.595,363.551,-83.768,-177.097,11.080,149.485
C07973=1131.599,363.304,-83.731,-177.100,11.078,149.485
C07974=1131.603,363.056,-83.695,-177.103,11.076,149.486
C07975=1131.606,362.844,-83.664,-177.107,11.073,149.486
C07976=1131.609,362.631,-83.633,-177.109,11.071,149.486
C07977=1131.613,362.418,-83.602,-177.113,11.069,149.486
C07978=1131.616,362.205,-83.571,-177.115,11.067,149.487
C07979=1131.619,361.993,-83.540,-177.118,11.066,149.487
C07980=1131.622,361.779,-83.509,-177.121,11.063,149.487
C07981=1131.626,361.567,-83.478,-177.124,11.061,149.487
C07982=1131.629,361.354,-83.447,-177.127,11.059,149.488
C07983=1131.633,361.107,-83.411,-177.131,11.056,149.488
C07984=1131.637,360.859,-83.375,-177.134,11.054,149.488
C07985=1131.640,360.612,-83.340,-177.137,11.052,149.488
C07986=1131.645,360.365,-83.303,-177.141,11.049,149.489
C07987=1131.648,360.117,-83.267,-177.144,11.047,149.489
C07988=1131.652,359.870,-83.232,-177.148,11.044,149.489
C07989=1131.656,359.622,-83.196,-177.151,11.042,149.489
C07990=1131.660,359.375,-83.159,-177.155,11.040,149.490
C07991=1131.663,359.128,-83.124,-177.158,11.037,149.490
C07992=1131.667,358.880,-83.088,-177.161,11.035,149.490
C07993=1131.671,358.633,-83.053,-177.164,11.032,149.490
C07994=1131.675,358.385,-83.016,-177.168,11.030,149.491
C07995=1131.679,358.139,-82.980,-177.171,11.028,149.491
C07996=1131.683,357.891,-82.945,-177.175,11.025,149.491
C07997=1131.686,357.644,-82.909,-177.179,11.022,149.492
C07998=1131.691,357.396,-82.873,-177.182,11.020,149.492
C07999=1131.694,357.148,-82.838,-177.186,11.018,149.492
C08000=1131.698,356.901,-82.802,-177.189,11.015,149.492
C08001=1131.702,356.653,-82.767,-177.193,11.013,149.493
C08002=1131.705,356.406,-82.731,-177.197,11.010,149.493
C08003=1131.710,356.159,-82.696,-177.200,11.007,149.493
C08004=1131.714,355.911,-82.660,-177.204,11.005,149.493
C08005=1131.718,355.664,-82.624,-177.207,11.003,149.494
C08006=1131.721,355.416,-82.589,-177.210,11.000,149.494
C08007=1131.725,355.169,-82.553,-177.214,10.997,149.494
C08008=1131.729,354.921,-82.518,-177.218,10.995,149.494
C08009=1131.733,354.674,-82.482,-177.221,10.992,149.495
C08010=1131.737,354.427,-82.447,-177.225,10.990,149.495
C08011=1131.740,354.179,-82.411,-177.229,10.987,149.495
C08012=1131.744,353.932,-82.376,-177.232,10.984,149.496
C08013=1131.748,353.684,-82.340,-177.236,10.982,149.496
C08014=1131.753,353.437,-82.304,-177.240,10.979,149.496
C08015=1131.756,353.190,-82.269,-177.243,10.977,149.496
C08016=1131.760,352.942,-82.234,-177.247,10.974,149.497
C08017=1131.764,352.694,-82.198,-177.250,10.971,149.497
C08018=1131.768,352.447,-82.163,-177.254,10.969,149.497
C08019=1131.772,352.200,-82.128,-177.257,10.966,149.497
C08020=1131.775,351.952,-82.092,-177.261,10.963,149.498
C08021=1131.779,351.704,-82.057,-177.265,10.961,149.498
C08022=1131.784,351.457,-82.022,-177.268,10.958,149.498
C08023=1131.787,351.210,-81.987,-177.272,10.955,149.498
C08024=1131.791,350.962,-81.952,-177.276,10.953,149.499
C08025=1131.795,350.714,-81.916,-177.280,10.950,149.499
C08026=1131.799,350.468,-81.882,-177.283,10.947,149.499
C08027=1131.802,350.220,-81.847,-177.287,10.945,149.499
C08028=1131.806,349.972,-81.811,-177.291,10.942,149.500
C08029=1131.810,349.725,-81.776,-177.294,10.940,149.500
C08030=1131.814,349.477,-81.741,-177.298,10.936,149.500
C08031=1131.818,349.264,-81.711,-177.301,10.935,149.501
C08032=1131.822,349.051,-81.681,-177.304,10.932,149.501
C08033=1131.824,348.838,-81.651,-177.307,10.930,149.501
C08034=1131.828,348.625,-81.620,-177.310,10.928,149.501
C08035=1131.832,348.413,-81.590,-177.312,10.926,149.501
C08036=1131.835,348.199,-81.561,-177.315,10.924,149.501
C08037=1131.838,347.986,-81.530,-177.318,10.921,149.501
C08038=1131.842,347.773,-81.500,-177.320,10.920,149.502
C08039=1131.845,347.526,-81.465,-177.324,10.917,149.502
C08040=1131.849,347.278,-81.430,-177.327,10.915,149.502
C08041=1131.853,347.030,-81.396,-177.330,10.912,149.502
C08042=1131.857,346.783,-81.360,-177.334,10.910,149.503
C08043=1131.862,346.535,-81.326,-177.337,10.907,149.503
C08044=1131.864,346.288,-81.291,-177.340,10.905,149.503
C08045=1131.868,346.040,-81.256,-177.343,10.902,149.503
C08046=1131.873,345.793,-81.221,-177.347,10.900,149.503
C08047=1131.877,345.545,-81.186,-177.350,10.897,149.504
C08048=1131.881,345.298,-81.151,-177.353,10.895,149.504
C08049=1131.884,345.051,-81.116,-177.356,10.892,149.504
C08050=1131.888,344.802,-81.081,-177.359,10.889,149.504
C08051=1131.893,344.555,-81.047,-177.363,10.887,149.504
C08052=1131.897,344.307,-81.012,-177.366,10.885,149.505
C08053=1131.900,344.060,-80.978,-177.369,10.882,149.505
C08054=1131.904,343.812,-80.943,-177.373,10.880,149.505
C08055=1131.909,343.565,-80.908,-177.376,10.877,149.505
C08056=1131.912,343.318,-80.873,-177.379,10.875,149.506
C08057=1131.916,343.070,-80.839,-177.382,10.872,149.506
C08058=1131.920,342.822,-80.804,-177.385,10.869,149.506
C08059=1131.924,342.575,-80.770,-177.389,10.867,149.506
C08060=1131.928,342.327,-80.735,-177.392,10.865,149.506
C08061=1131.933,342.080,-80.701,-177.395,10.862,149.506
C08062=1131.935,341.832,-80.666,-177.399,10.860,149.507
C08063=1131.940,341.585,-80.631,-177.401,10.858,149.507
C08064=1131.944,341.337,-80.597,-177.404,10.855,149.507
C08065=1131.948,341.090,-80.563,-177.408,10.853,149.507
C08066=1131.952,340.842,-80.528,-177.411,10.850,149.508
C08067=1131.956,340.594,-80.494,-177.414,10.848,149.508
C08068=1131.960,340.346,-80.459,-177.417,10.845,149.508
C08069=1131.964,340.099,-80.425,-177.421,10.843,149.508
C08070=1131.967,339.851,-80.390,-177.424,10.840,149.508
C08071=1131.972,339.604,-80.356,-177.427,10.838,149.509
C08072=1131.975,339.356,-80.322,-177.430,10.835,149.509
C08073=1131.980,339.108,-80.287,-177.434,10.833,149.509
C08074=1131.984,338.861,-80.253,-177.437,10.830,149.509
C08075=1131.988,338.613,-80.219,-177.440,10.828,149.509
C08076=1131.991,338.366,-80.185,-177.443,10.825,149.510
C08077=1131.995,338.118,-80.150,-177.447,10.823,149.510
C08078=1131.999,337.871,-80.116,-177.450,10.820,149.510
C08079=1132.003,337.623,-80.081,-177.453,10.817,149.510
C08080=1132.007,337.376,-80.047,-177.456,10.815,149.510
C08081=1132.012,337.128,-80.013,-177.460,10.812,149.511
C08082=1132.015,336.880,-79.979,-177.463,10.810,149.511
C08083=1132.020,336.632,-79.945,-177.466,10.807,149.511
C08084=1132.023,336.385,-79.911,-177.469,10.805,149.511
C08085=1132.027,336.137,-79.876,-177.472,10.802,149.511
C08086=1132.031,335.890,-79.842,-177.476,10.800,149.512
C08087=1132.034,335.676,-79.813,-177.478,10.798,149.512
C08088=1132.039,335.463,-79.784,-177.481,10.795,149.512
C08089=1132.041,335.250,-79.754,-177.484,10.793,149.512
C08090=1132.045,335.037,-79.725,-177.486,10.792,149.512
C08091=1132.048,334.824,-79.695,-177.489,10.789,149.512
C08092=1132.052,334.611,-79.666,-177.492,10.787,149.513
C08093=1132.055,334.398,-79.637,-177.495,10.785,149.513
C08094=1132.058,334.184,-79.608,-177.498,10.783,149.513
C08095=1132.062,333.937,-79.574,-177.501,10.780,149.513
C08096=1132.066,333.688,-79.540,-177.504,10.778,149.513
C08097=1132.070,333.441,-79.506,-177.507,10.775,149.513
C08098=1132.074,333.194,-79.472,-177.510,10.773,149.514
C08099=1132.078,332.945,-79.438,-177.514,10.770,149.514
C08100=1132.082,332.698,-79.404,-177.517,10.768,149.514
C08101=1132.086,332.451,-79.370,-177.520,10.765,149.514
C08102=1132.091,332.203,-79.337,-177.523,10.763,149.514
C08103=1132.094,331.955,-79.302,-177.527,10.760,149.515
C08104=1132.098,331.708,-79.269,-177.530,10.758,149.515
C08105=1132.102,331.460,-79.235,-177.533,10.755,149.515
C08106=1132.106,331.212,-79.201,-177.536,10.752,149.515
C08107=1132.110,330.965,-79.167,-177.540,10.750,149.515
C08108=1132.114,330.717,-79.134,-177.542,10.747,149.516
C08109=1132.118,330.470,-79.100,-177.546,10.745,149.516
C08110=1132.122,330.221,-79.067,-177.549,10.742,149.516
C08111=1132.126,329.974,-79.032,-177.552,10.740,149.516
C08112=1132.130,329.726,-78.999,-177.555,10.738,149.516
C08113=1132.134,329.479,-78.965,-177.558,10.735,149.517
C08114=1132.138,329.231,-78.932,-177.561,10.733,149.517
C08115=1132.142,328.983,-78.899,-177.565,10.731,149.517
C08116=1132.146,328.735,-78.864,-177.568,10.728,149.517
C08117=1132.151,328.488,-78.831,-177.571,10.725,149.517
C08118=1132.154,328.240,-78.797,-177.574,10.723,149.518
C08119=1132.158,327.992,-78.764,-177.577,10.720,149.518
C08120=1132.162,327.744,-78.730,-177.580,10.718,149.518
C08121=1132.166,327.497,-78.697,-177.584,10.715,149.518
C08122=1132.170,327.250,-78.663,-177.587,10.713,149.518
C08123=1132.174,327.001,-78.630,-177.590,10.710,149.518
C08124=1132.178,326.753,-78.597,-177.593,10.708,149.519
C08125=1132.182,326.506,-78.562,-177.597,10.705,149.519
C08126=1132.186,326.258,-78.529,-177.600,10.702,149.519
C08127=1132.191,326.011,-78.496,-177.603,10.700,149.519
C08128=1132.195,325.763,-78.463,-177.606,10.697,149.520
C08129=1132.198,325.514,-78.429,-177.609,10.695,149.520
C08130=1132.202,325.267,-78.395,-177.613,10.692,149.520
C08131=1132.206,325.020,-78.362,-177.616,10.690,149.520
C08132=1132.210,324.772,-78.329,-177.619,10.687,149.520
C08133=1132.215,324.524,-78.296,-177.622,10.685,149.520
C08134=1132.219,324.276,-78.263,-177.625,10.682,149.521
C08135=1132.223,324.029,-78.230,-177.629,10.680,149.521
C08136=1132.226,323.780,-78.196,-177.632,10.677,149.521
C08137=1132.230,323.533,-78.162,-177.634,10.675,149.521
C08138=1132.234,323.285,-78.129,-177.638,10.673,149.521
C08139=1132.238,323.038,-78.096,-177.641,10.670,149.522
C08140=1132.243,322.790,-78.063,-177.644,10.668,149.522
C08141=1132.246,322.543,-78.030,-177.647,10.665,149.522
C08142=1132.250,322.295,-77.997,-177.650,10.662,149.522
C08143=1132.254,322.081,-77.969,-177.653,10.660,149.522
C08144=1132.257,321.868,-77.940,-177.656,10.658,149.522
C08145=1132.261,321.654,-77.911,-177.658,10.656,149.523
C08146=1132.264,321.441,-77.883,-177.661,10.653,149.523
C08147=1132.268,321.228,-77.854,-177.664,10.651,149.523
C08148=1132.272,321.015,-77.825,-177.667,10.649,149.523
C08149=1132.274,320.801,-77.798,-177.669,10.647,149.523
C08150=1132.278,320.588,-77.769,-177.673,10.645,149.524
C08151=1132.282,320.340,-77.736,-177.675,10.643,149.524
C08152=1132.286,320.092,-77.703,-177.678,10.640,149.524
C08153=1132.290,319.844,-77.670,-177.682,10.638,149.524
C08154=1132.294,319.597,-77.637,-177.685,10.635,149.524
C08155=1132.298,319.349,-77.604,-177.688,10.633,149.524
C08156=1132.302,319.101,-77.571,-177.691,10.630,149.525
C08157=1132.306,318.853,-77.539,-177.694,10.627,149.525
C08158=1132.311,318.605,-77.505,-177.697,10.625,149.525
C08159=1132.314,318.358,-77.473,-177.701,10.622,149.525
C08160=1132.318,318.110,-77.440,-177.704,10.620,149.525
C08161=1132.322,317.863,-77.407,-177.707,10.617,149.526
C08162=1132.327,317.614,-77.374,-177.710,10.614,149.526
C08163=1132.330,317.367,-77.342,-177.713,10.612,149.526
C08164=1132.334,317.119,-77.308,-177.717,10.610,149.526
C08165=1132.339,316.871,-77.276,-177.720,10.607,149.526
C08166=1132.343,316.623,-77.243,-177.723,10.604,149.526
C08167=1132.346,316.376,-77.210,-177.726,10.602,149.527
C08168=1132.351,316.127,-77.178,-177.729,10.599,149.527
C08169=1132.355,315.879,-77.145,-177.732,10.597,149.527
C08170=1132.358,315.632,-77.112,-177.735,10.594,149.527
C08171=1132.363,315.384,-77.080,-177.738,10.592,149.527
C08172=1132.367,315.136,-77.046,-177.741,10.590,149.528
C08173=1132.370,314.889,-77.014,-177.744,10.587,149.528
C08174=1132.375,314.640,-76.981,-177.748,10.585,149.528
C08175=1132.379,314.393,-76.949,-177.751,10.582,149.528
C08176=1132.383,314.145,-76.917,-177.754,10.579,149.528
C08177=1132.387,313.897,-76.884,-177.757,10.577,149.529
C08178=1132.392,313.649,-76.851,-177.760,10.574,149.529
C08179=1132.395,313.402,-76.819,-177.763,10.572,149.529
C08180=1132.399,313.153,-76.786,-177.767,10.569,149.529
C08181=1132.403,312.906,-76.754,-177.770,10.567,149.529
C08182=1132.407,312.657,-76.721,-177.773,10.564,149.530
C08183=1132.411,312.410,-76.689,-177.776,10.561,149.530
C08184=1132.416,312.162,-76.657,-177.779,10.559,149.530
C08185=1132.420,311.914,-76.624,-177.783,10.556,149.530
C08186=1132.424,311.667,-76.592,-177.786,10.554,149.530
C08187=1132.428,311.418,-76.559,-177.789,10.551,149.530
C08188=1132.431,311.171,-76.527,-177.792,10.548,149.531
C08189=1132.436,310.923,-76.494,-177.795,10.546,149.531
C08190=1132.440,310.674,-76.462,-177.798,10.544,149.531
C08191=1132.444,310.427,-76.430,-177.801,10.542,149.531
C08192=1132.448,310.179,-76.398,-177.804,10.539,149.531
C08193=1132.452,309.931,-76.365,-177.807,10.536,149.531
C08194=1132.456,309.684,-76.333,-177.810,10.534,149.532
C08195=1132.460,309.435,-76.300,-177.813,10.531,149.532
C08196=1132.465,309.188,-76.269,-177.817,10.529,149.532
C08197=1132.469,308.940,-76.236,-177.820,10.526,149.532
C08198=1132.472,308.692,-76.204,-177.823,10.524,149.532
C08199=1132.476,308.478,-76.177,-177.825,10.522,149.533
C08200=1132.480,308.265,-76.149,-177.829,10.519,149.533
C08201=1132.483,308.052,-76.121,-177.831,10.517,149.533
C08202=1132.487,307.838,-76.093,-177.834,10.515,149.533
C08203=1132.490,307.624,-76.066,-177.836,10.513,149.533
C08204=1132.494,307.411,-76.038,-177.839,10.511,149.533
C08205=1132.497,307.198,-76.010,-177.842,10.508,149.534
C08206=1132.501,306.984,-75.982,-177.844,10.506,149.534
C08207=1132.505,306.737,-75.951,-177.847,10.504,149.534
C08208=1132.509,306.489,-75.919,-177.851,10.501,149.534
C08209=1132.513,306.240,-75.886,-177.854,10.499,149.534
C08210=1132.517,305.992,-75.855,-177.857,10.496,149.534
C08211=1132.522,305.745,-75.823,-177.860,10.493,149.535
C08212=1132.526,305.497,-75.791,-177.863,10.491,149.535
C08213=1132.529,305.249,-75.759,-177.867,10.488,149.535
C08214=1132.534,305.001,-75.727,-177.869,10.486,149.535
C08215=1132.538,304.753,-75.695,-177.873,10.483,149.535
C08216=1132.542,304.505,-75.663,-177.876,10.480,149.535
C08217=1132.546,304.257,-75.631,-177.879,10.478,149.536
C08218=1132.551,304.009,-75.599,-177.882,10.476,149.536
C08219=1132.554,303.761,-75.567,-177.885,10.473,149.536
C08220=1132.558,303.513,-75.535,-177.888,10.471,149.536
C08221=1132.563,303.266,-75.503,-177.891,10.468,149.536
C08222=1132.567,303.017,-75.472,-177.894,10.466,149.537
C08223=1132.570,302.769,-75.440,-177.897,10.463,149.537
C08224=1132.575,302.521,-75.409,-177.901,10.461,149.537
C08225=1132.579,302.273,-75.377,-177.903,10.458,149.537
C08226=1132.584,302.026,-75.345,-177.907,10.455,149.537
C08227=1132.588,301.778,-75.313,-177.910,10.453,149.537
C08228=1132.591,301.530,-75.281,-177.913,10.450,149.538
C08229=1132.596,301.282,-75.250,-177.916,10.447,149.538
C08230=1132.600,301.034,-75.219,-177.919,10.445,149.538
C08231=1132.605,300.786,-75.187,-177.922,10.442,149.538
C08232=1132.608,300.538,-75.155,-177.926,10.440,149.538
C08233=1132.612,300.290,-75.123,-177.928,10.438,149.539
C08234=1132.617,300.042,-75.092,-177.931,10.435,149.539
C08235=1132.620,299.794,-75.060,-177.935,10.433,149.539
C08236=1132.624,299.546,-75.029,-177.938,10.430,149.539
C08237=1132.628,299.299,-74.997,-177.941,10.428,149.539
C08238=1132.632,299.050,-74.966,-177.944,10.425,149.540
C08239=1132.637,298.802,-74.934,-177.947,10.423,149.540
C08240=1132.641,298.554,-74.902,-177.950,10.420,149.540
C08241=1132.646,298.306,-74.871,-177.953,10.417,149.540
C08242=1132.649,298.058,-74.839,-177.956,10.415,149.540
C08243=1132.654,297.810,-74.809,-177.960,10.412,149.540
C08244=1132.658,297.562,-74.777,-177.963,10.409,149.541
C08245=1132.661,297.314,-74.745,-177.966,10.407,149.541
C08246=1132.666,297.066,-74.714,-177.969,10.404,149.541
C08247=1132.670,296.818,-74.682,-177.972,10.403,149.541
C08248=1132.674,296.570,-74.652,-177.975,10.400,149.541
C08249=1132.678,296.322,-74.620,-177.978,10.397,149.542
C08250=1132.683,296.074,-74.589,-177.981,10.395,149.542
C08251=1132.686,295.826,-74.557,-177.984,10.392,149.542
C08252=1132.691,295.578,-74.526,-177.987,10.389,149.542
C08253=1132.695,295.330,-74.494,-177.990,10.387,149.542
C08254=1132.699,295.082,-74.464,-177.993,10.384,149.542
C08255=1132.703,294.868,-74.437,-177.996,10.382,149.542
C08256=1132.706,294.655,-74.410,-177.999,10.380,149.543
C08257=1132.710,294.442,-74.384,-178.001,10.378,149.543
C08258=1132.713,294.228,-74.356,-178.004,10.376,149.543
C08259=1132.717,294.015,-74.329,-178.007,10.373,149.543
C08260=1132.720,293.801,-74.302,-178.009,10.371,149.543
C08261=1132.723,293.587,-74.275,-178.012,10.369,149.543
C08262=1132.727,293.374,-74.249,-178.014,10.367,149.544
C08263=1132.731,293.125,-74.218,-178.018,10.364,149.544
C08264=1132.736,292.877,-74.187,-178.021,10.362,149.544
C08265=1132.740,292.629,-74.155,-178.024,10.359,149.544
C08266=1132.744,292.381,-74.124,-178.027,10.356,149.544
C08267=1132.748,292.134,-74.094,-178.030,10.354,149.545
C08268=1132.752,291.885,-74.062,-178.033,10.352,149.545
C08269=1132.757,291.638,-74.032,-178.036,10.350,149.545
C08270=1132.761,291.389,-74.000,-178.039,10.347,149.545
C08271=1132.765,291.141,-73.970,-178.042,10.344,149.545
C08272=1132.769,290.893,-73.938,-178.045,10.342,149.545
C08273=1132.773,290.645,-73.908,-178.049,10.339,149.546
C08274=1132.777,290.397,-73.877,-178.051,10.336,149.546
C08275=1132.781,290.149,-73.846,-178.054,10.334,149.546
C08276=1132.786,289.901,-73.815,-178.058,10.331,149.546
C08277=1132.789,289.652,-73.784,-178.061,10.328,149.546
C08278=1132.794,289.405,-73.753,-178.064,10.326,149.547
C08279=1132.798,289.157,-73.722,-178.067,10.323,149.547
C08280=1132.802,288.908,-73.691,-178.070,10.322,149.547
C08281=1132.806,288.661,-73.661,-178.073,10.319,149.547
C08282=1132.811,288.413,-73.630,-178.076,10.316,149.547
C08283=1132.815,288.164,-73.599,-178.079,10.314,149.547
C08284=1132.819,287.916,-73.569,-178.082,10.311,149.548
C08285=1132.823,287.668,-73.538,-178.085,10.308,149.548
C08286=1132.827,287.420,-73.507,-178.089,10.306,149.548
C08287=1132.831,287.172,-73.477,-178.091,10.303,149.548
C08288=1132.836,286.924,-73.446,-178.094,10.301,149.548
C08289=1132.840,286.676,-73.415,-178.098,10.298,149.549
C08290=1132.844,286.428,-73.385,-178.101,10.295,149.549
C08291=1132.848,286.180,-73.354,-178.104,10.293,149.549
C08292=1132.853,285.932,-73.323,-178.106,10.291,149.549
C08293=1132.856,285.684,-73.293,-178.110,10.289,149.549
C08294=1132.861,285.436,-73.262,-178.113,10.286,149.549
C08295=1132.865,285.188,-73.231,-178.116,10.283,149.549
C08296=1132.869,284.939,-73.201,-178.119,10.281,149.550
C08297=1132.874,284.691,-73.171,-178.122,10.278,149.550
C08298=1132.877,284.443,-73.140,-178.125,10.275,149.550
C08299=1132.882,284.195,-73.110,-178.128,10.273,149.550
C08300=1132.885,283.947,-73.079,-178.131,10.270,149.550
C08301=1132.890,283.699,-73.048,-178.134,10.267,149.551
C08302=1132.894,283.451,-73.018,-178.138,10.265,149.551
C08303=1132.899,283.203,-72.988,-178.140,10.263,149.551
C08304=1132.903,282.954,-72.957,-178.143,10.260,149.551
C08305=1132.907,282.706,-72.927,-178.146,10.258,149.551
C08306=1132.911,282.458,-72.896,-178.149,10.255,149.551
C08307=1132.915,282.210,-72.867,-178.153,10.253,149.552
C08308=1132.920,281.962,-72.836,-178.156,10.250,149.552
C08309=1132.923,281.714,-72.805,-178.159,10.248,149.552
C08310=1132.928,281.466,-72.775,-178.162,10.245,149.552
C08311=1132.931,281.252,-72.749,-178.165,10.242,149.553
C08312=1132.935,281.038,-72.723,-178.168,10.240,149.553
C08313=1132.939,280.825,-72.697,-178.171,10.237,149.553
C08314=1132.942,280.611,-72.671,-178.174,10.234,149.553
C08315=1132.946,280.397,-72.645,-178.177,10.233,149.553
C08316=1132.950,280.183,-72.619,-178.180,10.230,149.553
C08317=1132.953,279.970,-72.593,-178.183,10.228,149.554
C08318=1132.957,279.755,-72.567,-178.186,10.225,149.554
C08319=1132.961,279.508,-72.537,-178.190,10.222,149.554
C08320=1132.966,279.260,-72.506,-178.194,10.219,149.554
C08321=1132.970,279.011,-72.477,-178.197,10.217,149.554
C08322=1132.973,278.763,-72.446,-178.201,10.213,149.555
C08323=1132.978,278.515,-72.416,-178.204,10.211,149.555
C08324=1132.982,278.267,-72.386,-178.207,10.207,149.555
C08325=1132.986,278.019,-72.357,-178.211,10.205,149.555
C08326=1132.991,277.771,-72.326,-178.214,10.202,149.555
C08327=1132.995,277.522,-72.296,-178.218,10.199,149.556
C08328=1132.999,277.274,-72.267,-178.221,10.196,149.556
C08329=1133.003,277.026,-72.237,-178.224,10.194,149.556
C08330=1133.008,276.778,-72.207,-178.228,10.190,149.556
C08331=1133.012,276.530,-72.177,-178.231,10.188,149.556
C08332=1133.015,276.281,-72.147,-178.234,10.185,149.557
C08333=1133.020,276.033,-72.117,-178.237,10.183,149.557
C08334=1133.024,275.785,-72.087,-178.241,10.179,149.557
C08335=1133.028,275.537,-72.057,-178.244,10.176,149.557
C08336=1133.032,275.289,-72.028,-178.247,10.174,149.557
C08337=1133.036,275.041,-71.997,-178.250,10.171,149.557
C08338=1133.041,274.792,-71.967,-178.253,10.169,149.558
C08339=1133.045,274.544,-71.938,-178.256,10.166,149.558
C08340=1133.050,274.296,-71.909,-178.259,10.163,149.558
C08341=1133.053,274.048,-71.878,-178.262,10.161,149.558
C08342=1133.058,273.800,-71.849,-178.265,10.158,149.558
C08343=1133.062,273.552,-71.819,-178.269,10.154,149.558
C08344=1133.067,273.303,-71.789,-178.272,10.152,149.558
C08345=1133.071,273.055,-71.760,-178.274,10.150,149.559
C08346=1133.075,272.806,-71.730,-178.277,10.147,149.559
C08347=1133.079,272.559,-71.700,-178.280,10.144,149.559
C08348=1133.083,272.311,-71.671,-178.283,10.142,149.559
C08349=1133.087,272.062,-71.641,-178.286,10.139,149.559
C08350=1133.091,271.814,-71.612,-178.289,10.136,149.559
C08351=1133.096,271.566,-71.583,-178.292,10.133,149.559
C08352=1133.100,271.317,-71.553,-178.295,10.131,149.559
C08353=1133.104,271.069,-71.524,-178.298,10.128,149.559
C08354=1133.109,270.821,-71.494,-178.300,10.126,149.560
C08355=1133.113,270.572,-71.464,-178.303,10.123,149.560
C08356=1133.118,270.325,-71.435,-178.306,10.120,149.560
C08357=1133.122,270.077,-71.406,-178.309,10.118,149.560
C08358=1133.126,269.828,-71.376,-178.311,10.116,149.560
C08359=1133.130,269.580,-71.347,-178.314,10.113,149.560
C08360=1133.135,269.332,-71.317,-178.317,10.110,149.560
C08361=1133.139,269.083,-71.288,-178.319,10.108,149.560
C08362=1133.143,268.835,-71.258,-178.322,10.105,149.560
C08363=1133.147,268.587,-71.229,-178.325,10.103,149.561
C08364=1133.151,268.339,-71.199,-178.328,10.101,149.561
C08365=1133.156,268.090,-71.170,-178.331,10.098,149.561
C08366=1133.160,267.842,-71.140,-178.333,10.096,149.561
C08367=1133.163,267.629,-71.115,-178.335,10.094,149.561
C08368=1133.167,267.415,-71.091,-178.337,10.092,149.561
C08369=1133.171,267.201,-71.066,-178.339,10.090,149.561
C08370=1133.174,266.987,-71.040,-178.342,10.088,149.561
C08371=1133.178,266.773,-71.015,-178.344,10.085,149.561
C08372=1133.182,266.559,-70.990,-178.346,10.083,149.561
C08373=1133.185,266.345,-70.964,-178.348,10.081,149.561
C08374=1133.189,266.131,-70.939,-178.351,10.079,149.562
C08375=1133.194,265.883,-70.910,-178.352,10.077,149.561
C08376=1133.198,265.634,-70.880,-178.355,10.074,149.562
C08377=1133.202,265.387,-70.852,-178.358,10.072,149.562
C08378=1133.206,265.138,-70.823,-178.360,10.070,149.562
C08379=1133.211,264.890,-70.794,-178.363,10.067,149.562
C08380=1133.215,264.642,-70.764,-178.365,10.065,149.562
C08381=1133.219,264.393,-70.735,-178.367,10.063,149.562
C08382=1133.223,264.144,-70.706,-178.372,10.059,149.562
C08383=1133.228,263.897,-70.677,-178.376,10.056,149.563
C08384=1133.232,263.649,-70.648,-178.380,10.053,149.563
C08385=1133.236,263.400,-70.619,-178.384,10.050,149.563
C08386=1133.240,263.152,-70.590,-178.388,10.047,149.563
C08387=1133.245,262.904,-70.561,-178.392,10.043,149.564
C08388=1133.250,262.655,-70.532,-178.396,10.040,149.564
C08389=1133.253,262.407,-70.503,-178.399,10.037,149.564
C08390=1133.257,262.158,-70.474,-178.403,10.034,149.564
C08391=1133.262,261.911,-70.445,-178.407,10.031,149.565
C08392=1133.266,261.663,-70.416,-178.410,10.028,149.565
C08393=1133.270,261.414,-70.388,-178.414,10.024,149.565
C08394=1133.274,261.166,-70.358,-178.418,10.021,149.565
C08395=1133.279,260.918,-70.330,-178.422,10.018,149.565
C08396=1133.284,260.669,-70.300,-178.425,10.015,149.565
C08397=1133.287,260.421,-70.272,-178.429,10.012,149.566
C08398=1133.292,260.172,-70.244,-178.432,10.009,149.566
C08399=1133.297,259.924,-70.215,-178.435,10.005,149.566
C08400=1133.300,259.676,-70.186,-178.439,10.002,149.566
C08401=1133.305,259.427,-70.157,-178.442,10.000,149.566
C08402=1133.309,259.180,-70.129,-178.446,9.996,149.566
C08403=1133.313,258.931,-70.100,-178.449,9.993,149.567
C08404=1133.318,258.682,-70.071,-178.452,9.991,149.567
C08405=1133.322,258.435,-70.043,-178.456,9.987,149.567
C08406=1133.326,258.186,-70.014,-178.459,9.985,149.567
C08407=1133.330,257.938,-69.986,-178.462,9.981,149.567
C08408=1133.335,257.690,-69.957,-178.465,9.978,149.567
C08409=1133.339,257.441,-69.928,-178.468,9.976,149.567
C08410=1133.343,257.193,-69.900,-178.471,9.973,149.567
C08411=1133.348,256.945,-69.871,-178.474,9.970,149.568
C08412=1133.352,256.696,-69.843,-178.477,9.967,149.568
C08413=1133.357,256.448,-69.815,-178.480,9.963,149.568
C08414=1133.361,256.199,-69.787,-178.483,9.961,149.568
C08415=1133.365,255.951,-69.757,-178.486,9.958,149.568
C08416=1133.369,255.703,-69.729,-178.485,9.957,149.567
C08417=1133.374,255.454,-69.701,-178.484,9.957,149.567
C08418=1133.378,255.206,-69.673,-178.483,9.957,149.567
C08419=1133.382,254.957,-69.644,-178.482,9.956,149.566
C08420=1133.386,254.709,-69.615,-178.481,9.955,149.566
C08421=1133.391,254.461,-69.587,-178.482,9.954,149.566
C08422=1133.395,254.213,-69.559,-178.482,9.953,149.566
C08423=1133.399,253.999,-69.534,-178.483,9.952,149.566
C08424=1133.402,253.785,-69.510,-178.483,9.951,149.565
C08425=1133.406,253.571,-69.485,-178.484,9.950,149.565
C08426=1133.410,253.356,-69.461,-178.485,9.949,149.565
C08427=1133.414,253.142,-69.436,-178.486,9.948,149.565
C08428=1133.418,252.928,-69.412,-178.488,9.945,149.565
C08429=1133.422,252.714,-69.387,-178.490,9.944,149.566
C08430=1133.424,252.500,-69.363,-178.492,9.942,149.566
C08431=1133.429,252.252,-69.334,-178.494,9.940,149.566
C08432=1133.433,252.004,-69.306,-178.497,9.937,149.566
C08433=1133.438,251.756,-69.278,-178.500,9.935,149.566
C08434=1133.442,251.507,-69.249,-178.504,9.932,149.566
C08435=1133.447,251.259,-69.221,-178.508,9.929,149.567
C08436=1133.451,251.010,-69.193,-178.512,9.926,149.567
C08437=1133.454,250.762,-69.165,-178.516,9.922,149.567
C08438=1133.459,250.513,-69.136,-178.521,9.919,149.568
C08439=1133.463,250.265,-69.108,-178.526,9.915,149.568
C08440=1133.468,250.017,-69.080,-178.531,9.911,149.568
C08441=1133.472,249.768,-69.052,-178.537,9.907,149.569
C08442=1133.476,249.520,-69.024,-178.543,9.903,149.570
C08443=1133.481,249.271,-68.995,-178.549,9.898,149.570
C08444=1133.485,249.023,-68.968,-178.555,9.893,149.570
C08445=1133.489,248.775,-68.939,-178.562,9.888,149.571
C08446=1133.494,248.526,-68.912,-178.569,9.883,149.572
C08447=1133.499,248.278,-68.884,-178.576,9.878,149.572
C08448=1133.502,248.030,-68.856,-178.583,9.872,149.573
C08449=1133.507,247.782,-68.828,-178.591,9.866,149.574
C08450=1133.511,247.533,-68.801,-178.599,9.860,149.574
C08451=1133.515,247.285,-68.773,-178.604,9.856,149.575
C08452=1133.520,247.037,-68.744,-178.605,9.854,149.574
C08453=1133.524,246.787,-68.717,-178.606,9.852,149.574
C08454=1133.529,246.539,-68.689,-178.607,9.850,149.574
C08455=1133.533,246.290,-68.662,-178.608,9.848,149.574
C08456=1133.537,246.042,-68.634,-178.609,9.846,149.573
C08457=1133.541,245.795,-68.606,-178.610,9.844,149.573
C08458=1133.546,245.545,-68.579,-178.611,9.842,149.573
C08459=1133.551,245.297,-68.550,-178.612,9.840,149.573
C08460=1133.555,245.049,-68.523,-178.614,9.838,149.573
C08461=1133.559,244.800,-68.495,-178.616,9.836,149.573
C08462=1133.563,244.552,-68.467,-178.617,9.834,149.573
C08463=1133.568,244.304,-68.440,-178.618,9.832,149.573
C08464=1133.572,244.055,-68.412,-178.619,9.830,149.572
C08465=1133.576,243.807,-68.385,-178.621,9.827,149.572
C08466=1133.581,243.559,-68.357,-178.622,9.826,149.572
C08467=1133.585,243.310,-68.330,-178.624,9.823,149.572
C08468=1133.589,243.062,-68.302,-178.626,9.822,149.572
C08469=1133.593,242.812,-68.275,-178.627,9.819,149.572
C08470=1133.598,242.564,-68.246,-178.629,9.817,149.572
C08471=1133.603,242.316,-68.219,-178.631,9.815,149.572
C08472=1133.607,242.068,-68.192,-178.633,9.812,149.572
C08473=1133.611,241.819,-68.164,-178.635,9.810,149.572
C08474=1133.616,241.571,-68.136,-178.637,9.808,149.572
C08475=1133.620,241.322,-68.109,-178.638,9.806,149.572
C08476=1133.624,241.074,-68.081,-178.641,9.804,149.572
C08477=1133.629,240.825,-68.054,-178.643,9.801,149.572
C08478=1133.633,240.577,-68.027,-178.645,9.799,149.572
C08479=1133.637,240.363,-68.003,-178.647,9.798,149.572
C08480=1133.641,240.148,-67.979,-178.649,9.795,149.572
C08481=1133.644,239.935,-67.956,-178.650,9.793,149.572
C08482=1133.648,239.720,-67.932,-178.653,9.791,149.572
C08483=1133.652,239.506,-67.909,-178.655,9.789,149.572
C08484=1133.656,239.292,-67.885,-178.657,9.787,149.572
C08485=1133.659,239.078,-67.861,-178.658,9.785,149.572
C08486=1133.663,238.864,-67.838,-178.661,9.783,149.572
C08487=1133.667,238.616,-67.810,-178.663,9.780,149.572
C08488=1133.671,238.366,-67.783,-178.665,9.778,149.572
C08489=1133.676,238.118,-67.756,-178.668,9.775,149.572
C08490=1133.680,237.870,-67.728,-178.671,9.772,149.572
C08491=1133.685,237.622,-67.701,-178.673,9.770,149.572
C08492=1133.689,237.372,-67.674,-178.676,9.768,149.572
C08493=1133.694,237.124,-67.647,-178.679,9.765,149.573
C08494=1133.698,236.876,-67.619,-178.681,9.763,149.573
C08495=1133.703,236.628,-67.592,-178.684,9.760,149.573
C08496=1133.707,236.379,-67.565,-178.687,9.757,149.573
C08497=1133.711,236.130,-67.537,-178.690,9.754,149.573
C08498=1133.715,235.882,-67.510,-178.693,9.751,149.573
C08499=1133.720,235.634,-67.483,-178.696,9.749,149.573
C08500=1133.724,235.385,-67.456,-178.699,9.746,149.573
C08501=1133.729,235.137,-67.429,-178.702,9.743,149.573
C08502=1133.733,234.888,-67.402,-178.705,9.740,149.574
C08503=1133.738,234.639,-67.374,-178.708,9.737,149.574
C08504=1133.742,234.391,-67.348,-178.711,9.735,149.574
C08505=1133.746,234.143,-67.320,-178.714,9.732,149.574
C08506=1133.751,233.895,-67.293,-178.718,9.728,149.574
C08507=1133.755,233.646,-67.266,-178.721,9.726,149.574
C08508=1133.759,233.397,-67.239,-178.725,9.722,149.574
C08509=1133.763,233.149,-67.212,-178.727,9.719,149.575
C08510=1133.768,232.900,-67.185,-178.731,9.716,149.575
C08511=1133.773,232.652,-67.158,-178.734,9.713,149.575
C08512=1133.776,232.403,-67.132,-178.738,9.710,149.575
C08513=1133.781,232.155,-67.105,-178.742,9.706,149.575
C08514=1133.786,231.907,-67.078,-178.746,9.703,149.576
C08515=1133.790,231.658,-67.050,-178.749,9.700,149.576
C08516=1133.794,231.409,-67.024,-178.752,9.697,149.576
C08517=1133.799,231.160,-66.997,-178.756,9.694,149.576
C08518=1133.803,230.911,-66.970,-178.760,9.690,149.576
C08519=1133.807,230.663,-66.944,-178.763,9.687,149.576
C08520=1133.812,230.415,-66.917,-178.767,9.684,149.577
C08521=1133.817,230.166,-66.890,-178.771,9.679,149.577
C08522=1133.821,229.918,-66.863,-178.776,9.676,149.577
C08523=1133.825,229.669,-66.837,-178.780,9.672,149.577
C08524=1133.829,229.421,-66.810,-178.784,9.669,149.578
C08525=1133.834,229.172,-66.783,-178.787,9.665,149.578
C08526=1133.838,228.924,-66.757,-178.791,9.662,149.578
C08527=1133.843,228.675,-66.730,-178.796,9.658,149.578
C08528=1133.848,228.427,-66.703,-178.799,9.654,149.578
C08529=1133.852,228.178,-66.677,-178.803,9.651,149.578
C08530=1133.856,227.929,-66.651,-178.806,9.647,149.578
C08531=1133.860,227.681,-66.624,-178.810,9.644,149.579
C08532=1133.865,227.433,-66.597,-178.813,9.640,149.579
C08533=1133.869,227.184,-66.571,-178.817,9.637,149.579
C08534=1133.874,226.935,-66.544,-178.821,9.633,149.579
C08535=1133.877,226.721,-66.521,-178.824,9.630,149.579
C08536=1133.882,226.507,-66.499,-178.827,9.627,149.579
C08537=1133.885,226.292,-66.476,-178.830,9.624,149.579
C08538=1133.889,226.079,-66.453,-178.833,9.621,149.579
C08539=1133.893,225.864,-66.431,-178.836,9.617,149.579
C08540=1133.897,225.650,-66.408,-178.839,9.614,149.579
C08541=1133.901,225.435,-66.385,-178.842,9.612,149.579
C08542=1133.904,225.221,-66.362,-178.844,9.608,149.579
C08543=1133.909,224.973,-66.337,-178.848,9.605,149.579
C08544=1133.913,224.724,-66.310,-178.851,9.601,149.580
C08545=1133.918,224.475,-66.284,-178.854,9.598,149.580
C08546=1133.922,224.227,-66.258,-178.857,9.595,149.580
C08547=1133.926,223.978,-66.232,-178.860,9.592,149.580
C08548=1133.931,223.730,-66.205,-178.864,9.588,149.580
C08549=1133.935,223.481,-66.179,-178.867,9.584,149.580
C08550=1133.939,223.232,-66.153,-178.869,9.581,149.580
C08551=1133.944,222.984,-66.126,-178.873,9.578,149.580
C08552=1133.949,222.736,-66.101,-178.875,9.575,149.580
C08553=1133.953,222.487,-66.075,-178.878,9.571,149.580
C08554=1133.957,222.238,-66.048,-178.881,9.568,149.579
C08555=1133.962,221.989,-66.022,-178.884,9.565,149.580
C08556=1133.966,221.741,-65.997,-178.887,9.562,149.580
C08557=1133.970,221.492,-65.971,-178.890,9.558,149.579
C08558=1133.975,221.244,-65.944,-178.892,9.555,149.579
C08559=1133.980,220.995,-65.918,-178.895,9.552,149.579
C08560=1133.984,220.746,-65.893,-178.897,9.548,149.579
C08561=1133.988,220.498,-65.867,-178.900,9.545,149.579
C08562=1133.993,220.249,-65.840,-178.903,9.542,149.579
C08563=1133.998,220.001,-65.814,-178.906,9.538,149.579
C08564=1134.002,219.752,-65.789,-178.908,9.535,149.579
C08565=1134.006,219.503,-65.763,-178.911,9.532,149.579
C08566=1134.010,219.255,-65.737,-178.913,9.529,149.579
C08567=1134.015,219.007,-65.712,-178.915,9.527,149.579
C08568=1134.020,218.757,-65.685,-178.917,9.523,149.579
C08569=1134.024,218.509,-65.660,-178.920,9.520,149.579
C08570=1134.029,218.260,-65.634,-178.922,9.517,149.578
C08571=1134.033,218.011,-65.608,-178.925,9.514,149.578
C08572=1134.037,217.764,-65.582,-178.926,9.511,149.578
C08573=1134.041,217.515,-65.556,-178.929,9.508,149.578
C08574=1134.046,217.266,-65.531,-178.931,9.505,149.578
C08575=1134.051,217.018,-65.505,-178.933,9.502,149.578
C08576=1134.055,216.769,-65.479,-178.935,9.499,149.578
C08577=1134.060,216.520,-65.453,-178.937,9.497,149.578
C08578=1134.064,216.271,-65.427,-178.939,9.493,149.577
C08579=1134.069,216.023,-65.402,-178.941,9.491,149.577
C08580=1134.073,215.774,-65.376,-178.943,9.488,149.577
C08581=1134.077,215.525,-65.350,-178.945,9.485,149.577
C08582=1134.082,215.277,-65.326,-178.947,9.483,149.577
C08583=1134.087,215.028,-65.300,-178.949,9.479,149.577
C08584=1134.091,214.779,-65.274,-178.951,9.477,149.577
C08585=1134.095,214.530,-65.248,-178.952,9.474,149.577
C08586=1134.100,214.282,-65.223,-178.954,9.472,149.576
C08587=1134.104,214.033,-65.197,-178.956,9.469,149.576
C08588=1134.108,213.784,-65.172,-178.958,9.466,149.576
C08589=1134.113,213.536,-65.146,-178.960,9.464,149.576
C08590=1134.117,213.288,-65.120,-178.961,9.461,149.576
C08591=1134.125,212.878,-65.078,-178.963,9.457,149.575
C08592=1134.132,212.470,-65.037,-178.965,9.454,149.575
C08593=1134.139,212.061,-64.995,-178.967,9.450,149.575
C08594=1134.147,211.652,-64.953,-178.970,9.446,149.574
C08595=1134.167,210.518,-64.835,-178.074,7.690,148.906
C08596=1134.171,210.293,-64.813,-178.076,7.688,148.906
C08597=1134.175,210.066,-64.791,-178.079,7.686,148.906
C08598=1134.180,209.841,-64.768,-178.081,7.684,148.907
C08599=1134.184,209.570,-64.741,-178.084,7.681,148.907
C08600=1134.189,209.299,-64.713,-178.088,7.677,148.907
C08601=1134.194,209.029,-64.686,-178.091,7.674,148.907
C08602=1134.199,208.758,-64.659,-178.094,7.671,148.907
C08603=1134.204,208.510,-64.634,-178.097,7.669,148.907
C08604=1134.208,208.260,-64.610,-178.100,7.666,148.908
C08605=1134.213,208.012,-64.584,-178.102,7.664,148.908
C08606=1134.217,207.763,-64.559,-178.105,7.661,148.908
C08607=1134.222,207.515,-64.535,-178.108,7.659,148.908
C08608=1134.226,207.266,-64.510,-178.111,7.656,148.908
C08609=1134.231,207.017,-64.485,-178.114,7.653,148.908
C08610=1134.235,206.769,-64.461,-178.116,7.651,148.909
C08611=1134.240,206.519,-64.436,-178.119,7.648,148.909
C08612=1134.244,206.271,-64.411,-178.122,7.645,148.909
C08613=1134.249,206.022,-64.386,-178.125,7.642,148.909
C08614=1134.254,205.773,-64.361,-178.128,7.640,148.909
C08615=1134.258,205.525,-64.337,-178.130,7.638,148.910
C08616=1134.263,205.275,-64.312,-178.133,7.635,148.910
C08617=1134.267,205.027,-64.288,-178.136,7.632,148.910
C08618=1134.272,204.779,-64.263,-178.139,7.629,148.910
C08619=1134.276,204.530,-64.238,-178.142,7.627,148.910
C08620=1134.281,204.281,-64.214,-178.144,7.624,148.910
C08621=1134.285,204.033,-64.190,-178.148,7.622,148.911
C08622=1134.290,203.783,-64.165,-178.151,7.619,148.911
C08623=1134.294,203.535,-64.140,-178.153,7.616,148.911
C08624=1134.299,203.286,-64.116,-178.156,7.614,148.911
C08625=1134.303,203.037,-64.091,-178.159,7.611,148.911
C08626=1134.308,202.788,-64.067,-178.162,7.609,148.911
C08627=1134.313,202.540,-64.043,-178.165,7.606,148.912
C08628=1134.317,202.290,-64.018,-178.167,7.604,148.912
C08629=1134.322,202.042,-63.993,-178.170,7.601,148.912
C08630=1134.327,201.793,-63.969,-178.173,7.598,148.912
C08631=1134.330,201.544,-63.944,-178.176,7.596,148.912
C08632=1134.335,201.296,-63.920,-178.178,7.593,148.913
C08633=1134.340,201.047,-63.896,-178.182,7.591,148.913
C08634=1134.344,200.798,-63.871,-178.184,7.588,148.913
C08635=1134.349,200.549,-63.847,-178.187,7.585,148.913
C08636=1134.353,200.301,-63.822,-178.190,7.583,148.913
C08637=1134.358,200.052,-63.798,-178.193,7.581,148.914
C08638=1134.362,199.803,-63.773,-178.196,7.578,148.914
C08639=1134.367,199.555,-63.749,-178.199,7.575,148.914
C08640=1134.371,199.306,-63.725,-178.201,7.573,148.914
C08641=1134.376,199.057,-63.701,-178.204,7.570,148.914
C08642=1134.380,198.808,-63.677,-178.207,7.568,148.915
C08643=1134.385,198.559,-63.653,-178.210,7.565,148.915
C08644=1134.390,198.311,-63.628,-178.213,7.563,148.915
C08645=1134.394,198.062,-63.604,-178.216,7.560,148.915
C08646=1134.398,197.813,-63.580,-178.218,7.557,148.915
C08647=1134.403,197.564,-63.556,-178.221,7.555,148.916
C08648=1134.408,197.315,-63.532,-178.224,7.553,148.916
C08649=1134.412,197.067,-63.507,-178.227,7.550,148.916
C08650=1134.417,196.818,-63.483,-178.230,7.547,148.916
C08651=1134.421,196.568,-63.459,-178.232,7.545,148.916
C08652=1134.426,196.320,-63.435,-178.235,7.543,148.917
C08653=1134.430,196.072,-63.411,-178.238,7.540,148.917
C08654=1134.435,195.823,-63.388,-178.241,7.538,148.917
C08655=1134.440,195.574,-63.363,-178.244,7.535,148.917
C08656=1134.444,195.325,-63.339,-178.247,7.532,148.917
C08657=1134.449,195.076,-63.315,-178.250,7.530,148.918
C08658=1134.453,194.827,-63.291,-178.252,7.527,148.918
C08659=1134.457,194.579,-63.267,-178.255,7.525,148.918
C08660=1134.463,194.329,-63.243,-178.258,7.522,148.918
C08661=1134.467,194.081,-63.219,-178.260,7.520,148.918
C08662=1134.472,193.832,-63.196,-178.264,7.517,148.919
C08663=1134.476,193.584,-63.171,-178.267,7.515,148.919
C08664=1134.481,193.335,-63.147,-178.269,7.513,148.919
C08665=1134.485,193.085,-63.124,-178.272,7.510,148.919
C08666=1134.489,192.837,-63.100,-178.275,7.507,148.920
C08667=1134.495,192.588,-63.076,-178.278,7.505,148.920
C08668=1134.499,192.339,-63.052,-178.280,7.502,148.920
C08669=1134.504,192.090,-63.028,-178.284,7.500,148.920
C08670=1134.508,191.842,-63.004,-178.286,7.498,148.920
C08671=1134.513,191.593,-62.981,-178.289,7.495,148.921
C08672=1134.517,191.344,-62.957,-178.292,7.492,148.921
C08673=1134.522,191.095,-62.933,-178.295,7.491,148.921
C08674=1134.527,190.846,-62.910,-178.298,7.488,148.921
C08675=1134.531,190.598,-62.886,-178.301,7.485,148.922
C08676=1134.536,190.349,-62.863,-178.303,7.483,148.922
C08677=1134.540,190.100,-62.838,-178.306,7.481,148.922
C08678=1134.544,189.851,-62.815,-178.309,7.478,148.922
C08679=1134.549,189.602,-62.791,-178.311,7.476,148.922
C08680=1134.553,189.353,-62.767,-178.315,7.473,148.923
C08681=1134.558,189.104,-62.744,-178.318,7.470,148.923
C08682=1134.563,188.855,-62.721,-178.320,7.469,148.923
C08683=1134.567,188.607,-62.697,-178.323,7.466,148.923
C08684=1134.572,188.358,-62.673,-178.326,7.463,148.924
C08685=1134.576,188.109,-62.650,-178.329,7.461,148.924
C08686=1134.581,187.860,-62.626,-178.332,7.458,148.924
C08687=1134.585,187.611,-62.602,-178.335,7.456,148.924
C08688=1134.590,187.362,-62.579,-178.337,7.454,148.925
C08689=1134.595,187.113,-62.556,-178.340,7.451,148.925
C08690=1134.599,186.865,-62.532,-178.344,7.448,148.925
C08691=1134.604,186.616,-62.508,-178.346,7.446,148.925
C08692=1134.609,186.367,-62.485,-178.349,7.444,148.926
C08693=1134.614,186.118,-62.462,-178.351,7.442,148.926
C08694=1134.619,185.869,-62.438,-178.355,7.439,148.926
C08695=1134.623,185.620,-62.415,-178.357,7.436,148.926
C08696=1134.627,185.372,-62.392,-178.360,7.435,148.927
C08697=1134.632,185.123,-62.368,-178.363,7.432,148.927
C08698=1134.636,184.874,-62.345,-178.366,7.429,148.927
C08699=1134.641,184.625,-62.322,-178.368,7.427,148.927
C08700=1134.646,184.376,-62.298,-178.372,7.425,148.927
C08701=1134.651,184.127,-62.275,-178.374,7.423,148.928
C08702=1134.655,183.878,-62.252,-178.377,7.420,148.928
C08703=1134.660,183.609,-62.227,-178.380,7.417,148.928
C08704=1134.665,183.339,-62.201,-178.383,7.415,148.928
C08705=1134.670,183.070,-62.176,-178.387,7.412,148.929
C08706=1134.675,182.799,-62.151,-178.389,7.409,148.929
C08707=1134.679,182.551,-62.128,-178.392,7.407,148.929
C08708=1134.684,182.302,-62.105,-178.395,7.405,148.929
C08709=1134.689,182.053,-62.082,-178.398,7.403,148.930
C08710=1134.694,181.804,-62.058,-178.401,7.400,148.930
C08711=1134.697,181.555,-62.036,-178.404,7.397,148.930
C08712=1134.702,181.306,-62.012,-178.407,7.396,148.931
C08713=1134.707,181.057,-61.989,-178.409,7.393,148.931
C08714=1134.712,180.808,-61.966,-178.412,7.391,148.931
C08715=1134.716,180.560,-61.943,-178.415,7.388,148.931
C08716=1134.721,180.311,-61.920,-178.418,7.386,148.932
C08717=1134.726,180.062,-61.896,-178.420,7.384,148.932
C08718=1134.730,179.813,-61.874,-178.424,7.381,148.932
C08719=1134.735,179.564,-61.851,-178.426,7.379,148.932
C08720=1134.739,179.315,-61.828,-178.429,7.376,148.933
C08721=1134.744,179.067,-61.805,-178.432,7.375,148.933
C08722=1134.748,178.818,-61.782,-178.435,7.372,148.933
C08723=1134.753,178.569,-61.759,-178.438,7.369,148.933
C08724=1134.757,178.319,-61.737,-178.440,7.367,148.934
C08725=1134.762,178.070,-61.713,-178.444,7.365,148.934
C08726=1134.767,177.822,-61.690,-178.446,7.363,148.934
C08727=1134.771,177.573,-61.667,-178.449,7.360,148.934
C08728=1134.776,177.324,-61.645,-178.452,7.358,148.935
C08729=1134.780,177.075,-61.622,-178.455,7.356,148.935
C08730=1134.786,176.827,-61.599,-178.457,7.354,148.935
C08731=1134.790,176.578,-61.576,-178.460,7.351,148.935
C08732=1134.795,176.328,-61.554,-178.463,7.348,148.936
C08733=1134.799,176.079,-61.530,-178.466,7.347,148.936
C08734=1134.804,175.831,-61.508,-178.469,7.344,148.936
C08735=1134.809,175.582,-61.485,-178.472,7.342,148.937
C08736=1134.813,175.333,-61.462,-178.474,7.339,148.937
C08737=1134.818,175.083,-61.440,-178.477,7.337,148.937
C08738=1134.822,174.835,-61.417,-178.480,7.335,148.937
C08739=1134.827,174.586,-61.394,-178.483,7.333,148.938
C08740=1134.831,174.337,-61.372,-178.486,7.330,148.938
C08741=1134.836,174.088,-61.349,-178.488,7.328,148.938
C08742=1134.841,173.839,-61.327,-178.492,7.326,148.938
C08743=1134.846,173.590,-61.304,-178.494,7.324,148.939
C08744=1134.850,173.341,-61.281,-178.497,7.321,148.939
C08745=1134.855,173.092,-61.259,-178.500,7.319,148.939
C08746=1134.859,172.844,-61.236,-178.503,7.317,148.939
C08747=1134.864,172.594,-61.213,-178.506,7.314,148.940
C08748=1134.869,172.346,-61.191,-178.509,7.312,148.940
C08749=1134.873,172.097,-61.169,-178.511,7.309,148.940
C08750=1134.878,171.847,-61.146,-178.514,7.308,148.941
C08751=1134.883,171.599,-61.124,-178.517,7.305,148.941
C08752=1134.888,171.349,-61.101,-178.520,7.303,148.941
C08753=1134.892,171.101,-61.078,-178.523,7.301,148.941
C08754=1134.896,170.852,-61.057,-178.525,7.299,148.942
C08755=1134.901,170.603,-61.033,-178.529,7.296,148.942
C08756=1134.906,170.354,-61.012,-178.531,7.294,148.942
C08757=1134.911,170.105,-60.989,-178.534,7.291,148.943
C08758=1134.915,169.856,-60.966,-178.537,7.290,148.943
C08759=1134.920,169.607,-60.944,-178.540,7.287,148.943
C08760=1134.925,169.358,-60.922,-178.542,7.285,148.943
C08761=1134.929,169.110,-60.899,-178.546,7.283,148.944
C08762=1134.934,168.860,-60.877,-178.548,7.281,148.944
C08763=1134.939,168.611,-60.855,-178.551,7.278,148.944
C08764=1134.943,168.363,-60.832,-178.554,7.276,148.945
C08765=1134.948,168.113,-60.810,-178.557,7.275,148.945
C08766=1134.952,167.865,-60.789,-178.559,7.272,148.945
C08767=1134.957,167.615,-60.766,-178.562,7.270,148.946
C08768=1134.962,167.367,-60.744,-178.565,7.267,148.946
C08769=1134.966,167.118,-60.721,-178.568,7.265,148.946
C08770=1134.971,166.868,-60.699,-178.571,7.263,148.946
C08771=1134.976,166.619,-60.677,-178.574,7.261,148.947
C08772=1134.980,166.371,-60.654,-178.576,7.258,148.947
C08773=1134.985,166.122,-60.633,-178.579,7.257,148.947
C08774=1134.990,165.872,-60.610,-178.582,7.254,148.948
C08775=1134.995,165.624,-60.588,-178.585,7.252,148.948
C08776=1134.999,165.374,-60.566,-178.588,7.249,148.948
C08777=1135.004,165.126,-60.545,-178.591,7.248,148.948
C08778=1135.008,164.876,-60.523,-178.594,7.245,148.949
C08779=1135.013,164.628,-60.500,-178.596,7.243,148.949
C08780=1135.018,164.379,-60.478,-178.599,7.241,148.949
C08781=1135.023,164.130,-60.456,-178.602,7.239,148.950
C08782=1135.027,163.881,-60.434,-178.604,7.237,148.950
C08783=1135.032,163.632,-60.412,-178.608,7.234,148.950
C08784=1135.036,163.383,-60.390,-178.610,7.233,148.951
C08785=1135.041,163.134,-60.368,-178.613,7.230,148.951
C08786=1135.045,162.885,-60.346,-178.616,7.228,148.951
C08787=1135.051,162.636,-60.324,-178.619,7.225,148.952
C08788=1135.055,162.386,-60.302,-178.622,7.223,148.952
C08789=1135.060,162.138,-60.280,-178.624,7.222,148.952
C08790=1135.065,161.889,-60.259,-178.628,7.219,148.952
C08791=1135.069,161.640,-60.237,-178.630,7.217,148.953
C08792=1135.074,161.391,-60.215,-178.633,7.215,148.953
C08793=1135.078,161.142,-60.193,-178.636,7.213,148.953
C08794=1135.083,160.893,-60.171,-178.639,7.210,148.954
C08795=1135.087,160.644,-60.149,-178.641,7.208,148.954
C08796=1135.093,160.395,-60.128,-178.644,7.207,148.954
C08797=1135.097,160.146,-60.107,-178.647,7.204,148.955
C08798=1135.102,159.897,-60.084,-178.650,7.202,148.955
C08799=1135.107,159.648,-60.063,-178.653,7.199,148.955
C08800=1135.111,159.399,-60.041,-178.656,7.198,148.955
C08801=1135.116,159.150,-60.019,-178.658,7.196,148.956
C08802=1135.121,158.901,-59.997,-178.661,7.193,148.956
C08803=1135.125,158.651,-59.976,-178.664,7.191,148.956
C08804=1135.130,158.403,-59.954,-178.667,7.189,148.957
C08805=1135.134,158.153,-59.932,-178.670,7.187,148.957
C08806=1135.139,157.905,-59.911,-178.672,7.185,148.957
C08807=1135.145,157.635,-59.887,-178.675,7.183,148.958
C08808=1135.149,157.366,-59.864,-178.679,7.180,148.958
C08809=1135.155,157.098,-59.840,-178.681,7.178,148.958
C08810=1135.159,156.829,-59.818,-178.685,7.176,148.959
C08811=1135.164,156.580,-59.796,-178.687,7.174,148.959
C08812=1135.169,156.331,-59.774,-178.691,7.172,148.959
C08813=1135.174,156.081,-59.753,-178.693,7.170,148.960
C08814=1135.178,155.833,-59.731,-178.696,7.167,148.960
C08815=1135.183,155.584,-59.710,-178.699,7.165,148.960
C08816=1135.188,155.334,-59.688,-178.702,7.164,148.961
C08817=1135.192,155.086,-59.667,-178.705,7.161,148.961
C08818=1135.197,154.836,-59.646,-178.707,7.159,148.961
C08819=1135.201,154.587,-59.624,-178.710,7.157,148.962
C08820=1135.206,154.339,-59.602,-178.713,7.155,148.962
C08821=1135.212,154.089,-59.582,-178.716,7.153,148.962
C08822=1135.216,153.841,-59.560,-178.719,7.150,148.963
C08823=1135.221,153.591,-59.538,-178.722,7.149,148.963
C08824=1135.225,153.342,-59.517,-178.724,7.147,148.963
C08825=1135.230,153.094,-59.496,-178.728,7.144,148.964
C08826=1135.235,152.844,-59.475,-178.730,7.142,148.964
C08827=1135.239,152.595,-59.453,-178.733,7.141,148.964
C08828=1135.244,152.346,-59.432,-178.736,7.138,148.965
C08829=1135.249,152.097,-59.411,-178.739,7.136,148.965
C08830=1135.254,151.848,-59.390,-178.741,7.134,148.965
C08831=1135.258,151.599,-59.368,-178.744,7.132,148.966
C08832=1135.263,151.350,-59.347,-178.747,7.130,148.966
C08833=1135.268,151.101,-59.326,-178.750,7.128,148.966
C08834=1135.273,150.852,-59.305,-178.753,7.126,148.967
C08835=1135.278,150.603,-59.284,-178.755,7.124,148.967
C08836=1135.281,150.354,-59.262,-178.758,7.122,148.967
C08837=1135.287,150.104,-59.241,-178.761,7.120,148.968
C08838=1135.292,149.855,-59.220,-178.764,7.118,148.968
C08839=1135.297,149.607,-59.199,-178.767,7.116,148.968
C08840=1135.301,149.358,-59.178,-178.770,7.114,148.969
C08841=1135.305,149.108,-59.156,-178.772,7.112,148.969
C08842=1135.310,148.859,-59.135,-178.775,7.110,148.969
C08843=1135.315,148.610,-59.115,-178.778,7.107,148.970
C08844=1135.320,148.361,-59.093,-178.781,7.106,148.970
C08845=1135.325,148.112,-59.072,-178.784,7.104,148.970
C08846=1135.329,147.863,-59.052,-178.786,7.101,148.971
C08847=1135.334,147.613,-59.030,-178.789,7.099,148.971
C08848=1135.338,147.365,-59.009,-178.792,7.098,148.971
C08849=1135.343,147.116,-58.988,-178.795,7.095,148.972
C08850=1135.348,146.866,-58.967,-178.798,7.094,148.972
C08851=1135.353,146.617,-58.947,-178.801,7.092,148.972
C08852=1135.358,146.369,-58.925,-178.803,7.089,148.973
C08853=1135.362,146.120,-58.905,-178.806,7.087,148.973
C08854=1135.367,145.871,-58.884,-178.809,7.086,148.973
C08855=1135.372,145.621,-58.863,-178.812,7.084,148.974
C08856=1135.376,145.372,-58.842,-178.815,7.081,148.974
C08857=1135.381,145.123,-58.821,-178.818,7.080,148.975
C08858=1135.386,144.874,-58.800,-178.820,7.078,148.975
C08859=1135.391,144.625,-58.779,-178.823,7.075,148.975
C08860=1135.395,144.376,-58.759,-178.826,7.073,148.975
C08861=1135.400,144.127,-58.738,-178.829,7.072,148.976
C08862=1135.405,143.878,-58.718,-178.832,7.069,148.976
C08863=1135.410,143.628,-58.697,-178.835,7.068,148.977
C08864=1135.415,143.380,-58.676,-178.837,7.066,148.977
C08865=1135.420,143.130,-58.655,-178.840,7.064,148.977
C08866=1135.424,142.881,-58.635,-178.843,7.061,148.978
C08867=1135.429,142.633,-58.613,-178.846,7.060,148.978
C08868=1135.433,142.384,-58.593,-178.848,7.058,148.978
C08869=1135.437,142.134,-58.572,-178.851,7.056,148.979
C08870=1135.442,141.885,-58.551,-178.854,7.054,148.979
C08871=1135.447,141.636,-58.531,-178.857,7.052,148.979
C08872=1135.452,141.387,-58.510,-178.859,7.050,148.980
C08873=1135.456,141.138,-58.489,-178.862,7.048,148.980
C08874=1135.462,140.888,-58.469,-178.865,7.046,148.980
C08875=1135.466,140.639,-58.449,-178.868,7.044,148.981
C08876=1135.471,140.390,-58.428,-178.871,7.042,148.981
C08877=1135.476,140.141,-58.408,-178.874,7.040,148.982
C08878=1135.480,139.892,-58.387,-178.877,7.038,148.982
C08879=1135.485,139.643,-58.367,-178.880,7.036,148.982
C08880=1135.490,139.393,-58.346,-178.882,7.035,148.983
C08881=1135.494,139.144,-58.325,-178.885,7.032,148.983
C08882=1135.499,138.896,-58.305,-178.888,7.030,148.983
C08883=1135.505,138.647,-58.284,-178.891,7.028,148.984
C08884=1135.509,138.397,-58.265,-178.893,7.027,148.984
C08885=1135.514,138.148,-58.244,-178.896,7.025,148.984
C08886=1135.519,137.899,-58.223,-178.899,7.023,148.985
C08887=1135.524,137.650,-58.203,-178.902,7.021,148.985
C08888=1135.528,137.401,-58.183,-178.905,7.019,148.986
C08889=1135.533,137.151,-58.162,-178.907,7.017,148.986
C08890=1135.538,136.902,-58.142,-178.910,7.015,148.986
C08891=1135.542,136.654,-58.122,-178.913,7.013,148.987
C08892=1135.547,136.405,-58.101,-178.916,7.011,148.987
C08893=1135.552,136.155,-58.080,-178.918,7.010,148.987
C08894=1135.557,135.906,-58.061,-178.922,7.007,148.988
C08895=1135.561,135.657,-58.040,-178.924,7.005,148.988
C08896=1135.566,135.408,-58.020,-178.927,7.004,148.989
C08897=1135.572,135.159,-58.000,-178.930,7.002,148.989
C08898=1135.576,134.910,-57.980,-178.933,7.000,148.989
C08899=1135.580,134.661,-57.959,-178.936,6.998,148.990
C08900=1135.585,134.411,-57.940,-178.939,6.996,148.990
C08901=1135.590,134.162,-57.919,-178.941,6.994,148.991
C08902=1135.595,133.913,-57.898,-178.944,6.992,148.991
C08903=1135.600,133.663,-57.879,-178.946,6.991,148.991
C08904=1135.604,133.414,-57.858,-178.950,6.988,148.991
C08905=1135.609,133.166,-57.839,-178.952,6.986,148.992
C08906=1135.614,132.917,-57.819,-178.955,6.985,148.992
C08907=1135.618,132.668,-57.798,-178.958,6.983,148.993
C08908=1135.624,132.418,-57.778,-178.961,6.981,148.993
C08909=1135.628,132.169,-57.758,-178.964,6.979,148.993
C08910=1135.633,131.919,-57.738,-178.967,6.977,148.994
C08911=1135.638,131.651,-57.716,-178.969,6.975,148.994
C08912=1135.644,131.383,-57.695,-178.973,6.973,148.995
C08913=1135.649,131.114,-57.674,-178.975,6.971,148.995
C08914=1135.654,130.846,-57.651,-178.978,6.970,148.995
C08915=1135.659,130.596,-57.632,-178.981,6.967,148.996
C08916=1135.663,130.348,-57.611,-178.984,6.965,148.996
C08917=1135.668,130.098,-57.592,-178.987,6.964,148.997
C08918=1135.673,129.848,-57.572,-178.990,6.962,148.997
C08919=1135.678,129.600,-57.552,-178.992,6.960,148.997
C08920=1135.682,129.351,-57.532,-178.996,6.958,148.998
C08921=1135.687,129.102,-57.512,-178.998,6.956,148.998
C08922=1135.692,128.852,-57.492,-179.001,6.954,148.999
C08923=1135.697,128.603,-57.473,-179.004,6.953,148.999
C08924=1135.701,128.354,-57.453,-179.007,6.951,148.999
C08925=1135.706,128.105,-57.433,-179.009,6.949,149.000
C08926=1135.711,127.856,-57.413,-179.012,6.948,149.000
C08927=1135.716,127.607,-57.393,-179.015,6.945,149.001
C08928=1135.721,127.357,-57.374,-179.018,6.943,149.001
C08929=1135.725,127.108,-57.353,-179.021,6.942,149.001
C08930=1135.730,126.859,-57.334,-179.023,6.940,149.002
C08931=1135.735,126.610,-57.314,-179.026,6.938,149.002
C08932=1135.740,126.360,-57.295,-179.028,6.936,149.002
C08933=1135.744,126.111,-57.274,-179.032,6.934,149.003
C08934=1135.750,125.863,-57.255,-179.035,6.932,149.003
C08935=1135.754,125.613,-57.235,-179.037,6.931,149.003
C08936=1135.759,125.363,-57.216,-179.040,6.929,149.004
C08937=1135.764,125.115,-57.196,-179.043,6.927,149.004
C08938=1135.768,124.866,-57.177,-179.045,6.925,149.005
C08939=1135.773,124.616,-57.157,-179.048,6.924,149.005
C08940=1135.778,124.367,-57.137,-179.051,6.922,149.005
C08941=1135.783,124.118,-57.118,-179.054,6.920,149.006
C08942=1135.788,123.869,-57.098,-179.057,6.918,149.006
C08943=1135.792,123.619,-57.078,-179.060,6.916,149.007
C08944=1135.798,123.371,-57.059,-179.062,6.915,149.007
C08945=1135.802,123.121,-57.039,-179.065,6.913,149.007
C08946=1135.807,122.872,-57.020,-179.068,6.911,149.008
C08947=1135.812,122.623,-57.001,-179.071,6.909,149.008
C08948=1135.816,122.373,-56.981,-179.073,6.908,149.009
C08949=1135.821,122.125,-56.961,-179.077,6.905,149.009
C08950=1135.826,121.875,-56.941,-179.079,6.904,149.009
C08951=1135.830,121.626,-56.922,-179.082,6.902,149.010
C08952=1135.836,121.377,-56.903,-179.085,6.900,149.010
C08953=1135.840,121.128,-56.883,-179.088,6.899,149.011
C08954=1135.846,120.879,-56.864,-179.090,6.897,149.011
C08955=1135.850,120.629,-56.845,-179.093,6.895,149.011
C08956=1135.854,120.380,-56.825,-179.096,6.893,149.012
C08957=1135.860,120.131,-56.806,-179.098,6.892,149.012
C08958=1135.865,119.882,-56.787,-179.101,6.890,149.013
C08959=1135.870,119.633,-56.767,-179.104,6.888,149.013
C08960=1135.874,119.383,-56.748,-179.107,6.886,149.014
C08961=1135.879,119.134,-56.729,-179.110,6.884,149.014
C08962=1135.884,118.885,-56.709,-179.113,6.883,149.014
C08963=1135.888,118.636,-56.690,-179.115,6.881,149.015
C08964=1135.893,118.387,-56.671,-179.118,6.879,149.015
C08965=1135.898,118.137,-56.652,-179.121,6.878,149.016
C08966=1135.904,117.888,-56.633,-179.124,6.876,149.016
C08967=1135.908,117.639,-56.614,-179.127,6.875,149.017
C08968=1135.913,117.390,-56.594,-179.130,6.873,149.017
C08969=1135.918,117.140,-56.575,-179.132,6.871,149.017
C08970=1135.922,116.892,-56.556,-179.135,6.869,149.018
C08971=1135.927,116.642,-56.536,-179.138,6.868,149.018
C08972=1135.932,116.393,-56.518,-179.140,6.866,149.019
C08973=1135.937,116.143,-56.499,-179.144,6.864,149.019
C08974=1135.942,115.894,-56.479,-179.146,6.862,149.019
C08975=1135.946,115.645,-56.460,-179.149,6.860,149.020
C08976=1135.951,115.396,-56.441,-179.152,6.859,149.020
C08977=1135.957,115.146,-56.422,-179.155,6.857,149.021
C08978=1135.961,114.898,-56.403,-179.157,6.855,149.021
C08979=1135.966,114.648,-56.384,-179.160,6.854,149.021
C08980=1135.970,114.399,-56.365,-179.163,6.852,149.022
C08981=1135.976,114.149,-56.346,-179.166,6.850,149.022
C08982=1135.981,113.900,-56.327,-179.168,6.848,149.023
C08983=1135.985,113.651,-56.308,-179.171,6.847,149.023
C08984=1135.990,113.402,-56.288,-179.174,6.845,149.023
C08985=1135.995,113.152,-56.270,-179.177,6.843,149.024
C08986=1136.000,112.904,-56.251,-179.179,6.842,149.024
C08987=1136.004,112.655,-56.232,-179.182,6.840,149.025
C08988=1136.010,112.405,-56.213,-179.185,6.838,149.025
C08989=1136.014,112.156,-56.194,-179.187,6.837,149.025
C08990=1136.019,111.906,-56.176,-179.191,6.835,149.026
C08991=1136.024,111.657,-56.157,-179.193,6.834,149.027
C08992=1136.029,111.408,-56.137,-179.196,6.832,149.027
C08993=1136.033,111.159,-56.119,-179.199,6.830,149.027
C08994=1136.039,110.910,-56.100,-179.202,6.829,149.028
C08995=1136.043,110.660,-56.082,-179.204,6.827,149.028
C08996=1136.048,110.411,-56.062,-179.207,6.825,149.029
C08997=1136.053,110.163,-56.044,-179.210,6.824,149.029
C08998=1136.058,109.912,-56.025,-179.213,6.822,149.029
C08999=1136.063,109.664,-56.006,-179.215,6.820,149.030
C09000=1136.067,109.414,-55.988,-179.218,6.819,149.030
C09001=1136.072,109.165,-55.968,-179.221,6.816,149.031
C09002=1136.077,108.916,-55.950,-179.224,6.814,149.031
C09003=1136.082,108.666,-55.931,-179.227,6.813,149.031
C09004=1136.087,108.417,-55.913,-179.230,6.811,149.032
C09005=1136.092,108.169,-55.894,-179.233,6.810,149.032
C09006=1136.097,107.918,-55.875,-179.235,6.808,149.033
C09007=1136.101,107.669,-55.857,-179.238,6.806,149.033
C09008=1136.107,107.420,-55.838,-179.240,6.806,149.034
C09009=1136.111,107.170,-55.819,-179.243,6.804,149.034
C09010=1136.116,106.922,-55.801,-179.246,6.802,149.035
C09011=1136.121,106.672,-55.782,-179.249,6.801,149.035
C09012=1136.125,106.423,-55.763,-179.251,6.799,149.035
C09013=1136.130,106.174,-55.745,-179.254,6.797,149.036
C09014=1136.136,105.925,-55.727,-179.257,6.796,149.036
C09015=1136.140,105.656,-55.706,-179.261,6.793,149.037
C09016=1136.146,105.388,-55.686,-179.263,6.792,149.037
C09017=1136.151,105.119,-55.667,-179.266,6.790,149.038
C09018=1136.156,104.851,-55.647,-179.269,6.788,149.038
C09019=1136.161,104.602,-55.628,-179.272,6.787,149.038
C09020=1136.166,104.352,-55.610,-179.275,6.785,149.039
C09021=1136.171,104.103,-55.592,-179.277,6.784,149.040
C09022=1136.176,103.854,-55.573,-179.280,6.782,149.040
C09023=1136.181,103.605,-55.554,-179.283,6.780,149.040
C09024=1136.185,103.355,-55.536,-179.286,6.779,149.041
C09025=1136.190,103.106,-55.518,-179.288,6.777,149.041
C09026=1136.196,102.857,-55.499,-179.291,6.775,149.042
C09027=1136.200,102.608,-55.481,-179.294,6.774,149.042
C09028=1136.205,102.358,-55.462,-179.297,6.772,149.042
C09029=1136.210,102.109,-55.444,-179.300,6.771,149.043
C09030=1136.215,101.860,-55.426,-179.303,6.769,149.043
C09031=1136.220,101.610,-55.408,-179.305,6.767,149.044
C09032=1136.225,101.360,-55.390,-179.308,6.766,149.044
C09033=1136.229,101.112,-55.371,-179.311,6.764,149.045
C09034=1136.234,100.863,-55.353,-179.313,6.762,149.045
C09035=1136.239,100.614,-55.335,-179.316,6.762,149.046
C09036=1136.244,100.364,-55.317,-179.318,6.760,149.046
C09037=1136.249,100.114,-55.298,-179.321,6.758,149.046
C09038=1136.254,99.865,-55.280,-179.324,6.757,149.047
C09039=1136.259,99.616,-55.262,-179.327,6.755,149.047
C09040=1136.264,99.367,-55.244,-179.330,6.754,149.048
C09041=1136.269,99.118,-55.226,-179.333,6.752,149.048
C09042=1136.273,98.869,-55.207,-179.335,6.750,149.049
C09043=1136.277,98.619,-55.189,-179.338,6.749,149.049
C09044=1136.282,98.370,-55.171,-179.341,6.747,149.050
C09045=1136.287,98.121,-55.153,-179.343,6.745,149.050
C09046=1136.293,97.871,-55.134,-179.347,6.744,149.051
C09047=1136.298,97.622,-55.116,-179.349,6.742,149.051
C09048=1136.303,97.373,-55.098,-179.352,6.741,149.051
C09049=1136.307,97.123,-55.080,-179.354,6.740,149.052
C09050=1136.312,96.874,-55.062,-179.357,6.738,149.052
C09051=1136.317,96.625,-55.044,-179.360,6.736,149.053
C09052=1136.322,96.375,-55.027,-179.363,6.735,149.053
C09053=1136.327,96.126,-55.009,-179.366,6.733,149.054
C09054=1136.332,95.877,-54.991,-179.368,6.732,149.054
C09055=1136.337,95.627,-54.973,-179.371,6.730,149.055
C09056=1136.342,95.378,-54.955,-179.374,6.728,149.055
C09057=1136.347,95.129,-54.937,-179.377,6.727,149.055
C09058=1136.352,94.880,-54.919,-179.379,6.725,149.056
C09059=1136.356,94.630,-54.901,-179.382,6.724,149.056
C09060=1136.361,94.381,-54.883,-179.385,6.723,149.057
C09061=1136.366,94.132,-54.865,-179.388,6.721,149.057
C09062=1136.371,93.882,-54.847,-179.390,6.720,149.058
C09063=1136.376,93.633,-54.829,-179.393,6.718,149.058
C09064=1136.381,93.383,-54.812,-179.396,6.716,149.059
C09065=1136.386,93.134,-54.794,-179.399,6.715,149.059
C09066=1136.391,92.885,-54.776,-179.402,6.713,149.060
C09067=1136.396,92.635,-54.758,-179.404,6.712,149.060
C09068=1136.401,92.386,-54.740,-179.407,6.711,149.060
C09069=1136.405,92.137,-54.723,-179.409,6.709,149.061
C09070=1136.410,91.888,-54.705,-179.412,6.707,149.061
C09071=1136.415,91.638,-54.688,-179.415,6.706,149.062
C09072=1136.420,91.389,-54.670,-179.418,6.704,149.062
C09073=1136.425,91.140,-54.652,-179.421,6.703,149.063
C09074=1136.430,90.891,-54.634,-179.424,6.701,149.063
C09075=1136.435,90.641,-54.616,-179.426,6.699,149.064
C09076=1136.440,90.392,-54.599,-179.428,6.699,149.064
C09077=1136.444,90.143,-54.581,-179.431,6.697,149.064
C09078=1136.449,89.893,-54.564,-179.434,6.696,149.065
C09079=1136.454,89.644,-54.546,-179.437,6.694,149.066
C09080=1136.459,89.395,-54.528,-179.440,6.692,149.066
C09081=1136.464,89.145,-54.511,-179.443,6.691,149.066
C09082=1136.469,88.896,-54.493,-179.445,6.689,149.067
C09083=1136.473,88.647,-54.475,-179.448,6.688,149.067
C09084=1136.479,88.397,-54.458,-179.451,6.687,149.068
C09085=1136.484,88.148,-54.440,-179.453,6.685,149.068
C09086=1136.489,87.898,-54.423,-179.456,6.683,149.069
C09087=1136.494,87.649,-54.405,-179.459,6.682,149.069
C09088=1136.498,87.399,-54.388,-179.462,6.680,149.070
C09089=1136.503,87.150,-54.370,-179.464,6.679,149.070
C09090=1136.508,86.901,-54.352,-179.467,6.678,149.071
C09091=1136.513,86.651,-54.335,-179.470,6.676,149.071
C09092=1136.517,86.402,-54.317,-179.473,6.675,149.072
C09093=1136.523,86.153,-54.300,-179.475,6.673,149.072
C09094=1136.528,85.904,-54.283,-179.478,6.671,149.072
C09095=1136.533,85.654,-54.265,-179.481,6.671,149.073
C09096=1136.538,85.406,-54.248,-179.483,6.669,149.073
C09097=1136.543,85.156,-54.231,-179.486,6.668,149.074
C09098=1136.548,84.906,-54.213,-179.489,6.666,149.074
C09099=1136.552,84.657,-54.196,-179.492,6.664,149.075
C09100=1136.557,84.407,-54.179,-179.495,6.663,149.075
C09101=1136.562,84.158,-54.161,-179.497,6.662,149.076
C09102=1136.567,83.909,-54.144,-179.500,6.660,149.076
C09103=1136.572,83.659,-54.126,-179.503,6.659,149.077
C09104=1136.577,83.410,-54.109,-179.505,6.657,149.077
C09105=1136.582,83.161,-54.093,-179.508,6.656,149.078
C09106=1136.587,82.912,-54.075,-179.511,6.655,149.078
C09107=1136.592,82.662,-54.057,-179.513,6.653,149.079
C09108=1136.597,82.412,-54.041,-179.516,6.652,149.079
